	(*X*)
	Quota_Prelievo_Falda_X : LREAL;
	Quota_Deposito_Falda_SuCatastaPallet_X : LREAL;
	Quota_Deposito_Falda_SuPiazzola_X : LREAL;
	Quota_Fuori_Ingombro_X : LREAL;	
	
	(*Y*)
	Quota_Prelievo_Falda_Y 					: LREAL;
	Quota_Deposito_Falda_SuCatastaPallet_Y 	: LREAL;
	Quota_Deposito_Falda_SuPiazzola_Y		: LREAL;
	
	Quota_Fuori_Ingombro_Y					: LREAL;
	
	(*Z*)
	Quota_StartLenta_Prelievo_Falda_Z 					: LREAL;
	Quota_Prelievo_Falda_Z 								: LREAL;
	Quota_StartLenta_Deposito_Falda_SuPiazzola_Z 		: LREAL; //Se non si utilizza il tasteggio in fase di deposito si utilizza questa quota come quota di rilascio!!!
	Quota_Deposito_Falda_SuPiazzola_Z					: LREAL;
	Quota_StartLenta_Deposito_Falda_SuCatastaPallet_Z	: LREAL;
	Quota_Deposito_Falda_SuCatastaPallet_Z				: LREAL;
	QUota_Fuori_Ingombro_Falda_Z 						: LREAL;
	Quota_Attesa_Caduta_Falda_Z							: LREAL;
	
	(*k*)
	//Quota_Apertura_Prelievo_Falda_K : LREAL;
	//Quota_Chiusura_Prelievo_Falda_K : LREAL;
	//Quota_Apertura_Deposito_Falda_K : LREAL;
		
	(*J*)
	Quota_Rotazione_Prelievo_Falda 			: LREAL;
	Quota_Rotazione_Deposito_Falda 			: LREAL;
	
END_VAR
VAR_OUTPUT
	Inizializzato : BOOL;
END_VAR
VAR
	;	
END_VAR

(*
PRELIEVO FALDA:
1- Programma asse X per raggiungere magazzino falde da quota attuale in direzione X
2- Programma asse Y per raggiungere magazzino falde da quota attuale in direzione Y
3- Programma asse J per raggiungere l'angolo di rotazione richiesto
4- Programma asse K per raggiungere la quota di apertura pinza 
5- Programma asse Z per raggiungere la quota di cambio velocità in direzione Z (si passerà da veloce a lenta + tastatori disabilitati) in VELOCE
6- Programma asse Z in cui si effettua la traslazione in LENTA in direzione Z fino tocco dei tastatori
7- Programma asse K per raggiungere la quota di chiusura pinza !!!! PREVISTO MA NON UTILIZZATO !!!!!!

DEPOSITO FALDA:
8- Programma asse Z per raggiungere la quota di "Attesa caduta Falda" 
9- Programma asse Z per raggiungere la quota di "Fuori Ingombro" ostacoli 
10- Programma asse X per raggiungere la quota di deposito falda da quota attuale in direzione X; puù essere sul pallet in catasta(ciclo vuoti) o pallet su piazzola
11- Programma asse Y per posizione la quota di deposito falda da quota attuale in direzione Y
12: 
12.1- Programma asse Z per raggiungere la quota di rilascio falda in direzione Z su PIAZZOLA
12.2- Programma asse Z Z in cui si effettua la traslazione in LENTA in direzione Z fino tocco dei tastatori su CATASTA VUOTI

*)
Inizializzato := FALSE;
(*************************************************************************************************************************************)
(******************************************************  ASSE X **********************************************************************)
(*************************************************************************************************************************************)
(* Programma 51 Asse X : Traslazione Verso Postazione di Prelievo Pacco*)
Programma_X[X_PosPrelievoFalda].ID 					:= X_PosPrelievoFalda;
Programma_X[X_PosPrelievoFalda].Quota_Destinazione	:= Quota_Prelievo_Falda_X;
Programma_X[X_PosPrelievoFalda].Velocita			:= X_Par.Vel_Vuoto;
Programma_X[X_PosPrelievoFalda].Accelerazione		:= X_Par.Acc_Vuoto;
Programma_X[X_PosPrelievoFalda].Decelerazione		:= X_Par.Dec_Vuoto;
Programma_X[X_PosPrelievoFalda].Jerk				:= X_Par.Jerk_Vuoto;

(* Programma 52 Asse X : Traslazione Verso Postazione di deposito Falda su catasta vuoti*)
Programma_X[X_PosDepositoSuCatastaFalda].ID 					:= X_PosDepositoSuCatastaFalda;
Programma_X[X_PosDepositoSuCatastaFalda].Quota_Destinazione	:= Quota_Deposito_Falda_SuCatastaPallet_X;
Programma_X[X_PosDepositoSuCatastaFalda].Velocita			:= X_Par.Vel_Vuoto;
Programma_X[X_PosDepositoSuCatastaFalda].Accelerazione		:= X_Par.Acc_Vuoto;
Programma_X[X_PosDepositoSuCatastaFalda].Decelerazione		:= X_Par.Dec_Vuoto;
Programma_X[X_PosDepositoSuCatastaFalda].Jerk				:= X_Par.Jerk_Vuoto;

(* Programma 53 Asse X : Traslazione a quota di deposito Falda su piazzola*)
Programma_X[X_PosDepositoFalda].ID 					:= X_PosDepositoFalda;
Programma_X[X_PosDepositoFalda].Quota_Destinazione	:= Quota_Deposito_Falda_SuPiazzola_X;
Programma_X[X_PosDepositoFalda].Velocita			:= X_Par.Vel_Vuoto;
Programma_X[X_PosDepositoFalda].Accelerazione		:= X_Par.Acc_Vuoto;
Programma_X[X_PosDepositoFalda].Decelerazione		:= X_Par.Dec_Vuoto;
Programma_X[X_PosDepositoFalda].Jerk				:= X_Par.Jerk_Vuoto;

(* Programma 56 Asse Y : Traslazione a quota di riposo a Vuoto *)
Programma_X[X_PosFuoriIngombroVuotoFalda].ID 					:= X_PosFuoriIngombroVuotoFalda;
Programma_X[X_PosFuoriIngombroVuotoFalda].Quota_Destinazione	:= Quota_Fuori_Ingombro_X;
Programma_X[X_PosFuoriIngombroVuotoFalda].Velocita			:= X_Par.Vel_Vuoto;
Programma_X[X_PosFuoriIngombroVuotoFalda].Accelerazione		:= X_Par.Acc_Vuoto;
Programma_X[X_PosFuoriIngombroVuotoFalda].Decelerazione		:= X_Par.Dec_Vuoto;
Programma_X[X_PosFuoriIngombroVuotoFalda].Jerk				:= X_Par.Jerk_Vuoto;

(*************************************************************************************************************************************)
(******************************************************  ASSE Y **********************************************************************)
(*************************************************************************************************************************************)
(* Programma 51 Asse Y : Traslazione a quota di Prelievo Falda*)
Programma_Y[Y_PosPrelievoFalda].ID 					:= Y_PosPrelievoFalda;
Programma_Y[Y_PosPrelievoFalda].Quota_Destinazione	:= Quota_Prelievo_Falda_Y;
Programma_Y[Y_PosPrelievoFalda].Velocita			:= Y_Par.Vel_Vuoto;
Programma_Y[Y_PosPrelievoFalda].Accelerazione		:= Y_Par.Acc_Vuoto;
Programma_Y[Y_PosPrelievoFalda].Decelerazione		:= Y_Par.Dec_Vuoto;
Programma_Y[Y_PosPrelievoFalda].Jerk				:= Y_Par.Jerk_Vuoto;

(* Programma 52 Asse Y : Traslazione a quota di Deposito Falda su catasta vuoti*)
Programma_Y[Y_PosDepositoSuCatastaFalda].ID 					:= Y_PosDepositoSuCatastaFalda;
Programma_Y[Y_PosDepositoSuCatastaFalda].Quota_Destinazione	:= Quota_Deposito_Falda_SuCatastaPallet_Y;
Programma_Y[Y_PosDepositoSuCatastaFalda].Velocita			:= Y_Par.Vel_Vuoto;
Programma_Y[Y_PosDepositoSuCatastaFalda].Accelerazione		:= Y_Par.Acc_Vuoto;
Programma_Y[Y_PosDepositoSuCatastaFalda].Decelerazione		:= Y_Par.Dec_Vuoto;
Programma_Y[Y_PosDepositoSuCatastaFalda].Jerk				:= Y_Par.Jerk_Vuoto;

(* Programma 53 Asse Y : Traslazione a quota di Deposito Falda su piazzola*)
Programma_Y[Y_PosDepositoFalda].ID 					:= Y_PosDepositoFalda;
Programma_Y[Y_PosDepositoFalda].Quota_Destinazione	:= Quota_Deposito_Falda_SuPiazzola_Y;
Programma_Y[Y_PosDepositoFalda].Velocita			:= Y_Par.Vel_Vuoto;
Programma_Y[Y_PosDepositoFalda].Accelerazione		:= Y_Par.Acc_Vuoto;
Programma_Y[Y_PosDepositoFalda].Decelerazione		:= Y_Par.Dec_Vuoto;
Programma_Y[Y_PosDepositoFalda].Jerk				:= Y_Par.Jerk_Vuoto;

(* Programma 56 Asse Y : Traslazione a quota di riposo a Vuoto *)
Programma_Y[Y_PosFuoriIngombroVuotoFalda].ID 					:= Y_PosFuoriIngombroVuotoFalda;
Programma_Y[Y_PosFuoriIngombroVuotoFalda].Quota_Destinazione	:= Quota_Fuori_Ingombro_Y;
Programma_Y[Y_PosFuoriIngombroVuotoFalda].Velocita			:= Y_Par.Vel_Vuoto;
Programma_Y[Y_PosFuoriIngombroVuotoFalda].Accelerazione		:= Y_Par.Acc_Vuoto;
Programma_Y[Y_PosFuoriIngombroVuotoFalda].Decelerazione		:= Y_Par.Dec_Vuoto;
Programma_Y[Y_PosFuoriIngombroVuotoFalda].Jerk				:= Y_Par.Jerk_Vuoto;

(* Programma 66 Asse Y : Traslazione a quota di riposo con carico*)
Programma_Y[Y_PosFuoriIngombroCaricoFalda].ID 					:= Y_PosFuoriIngombroCaricoFalda;
Programma_Y[Y_PosFuoriIngombroCaricoFalda].Quota_Destinazione	:= Quota_Fuori_Ingombro_Y;
Programma_Y[Y_PosFuoriIngombroCaricoFalda].Velocita			:= Y_Par.Vel_Carico;
Programma_Y[Y_PosFuoriIngombroCaricoFalda].Accelerazione		:= Y_Par.Acc_Carico;
Programma_Y[Y_PosFuoriIngombroCaricoFalda].Decelerazione		:= Y_Par.Dec_Carico;
Programma_Y[Y_PosFuoriIngombroCaricoFalda].Jerk				:= Y_Par.Jerk_Carico;

(*************************************************************************************************************************************)
(******************************************************  ASSE Z **********************************************************************)
(*************************************************************************************************************************************)

(* Programma 51 Asse Z : Traslazione veloce fino alla quota ammessa in fase di Prelievo Falda*)
Programma_Z[Z_PosStartLentaPrelievoFalda].ID 					:= Z_PosStartLentaPrelievoFalda;
Programma_Z[Z_PosStartLentaPrelievoFalda].Quota_Destinazione	:= Quota_StartLenta_Prelievo_Falda_Z;
Programma_Z[Z_PosStartLentaPrelievoFalda].Velocita			:= Z_Par.Vel_Vuoto;
Programma_Z[Z_PosStartLentaPrelievoFalda].Accelerazione		:= Z_Par.Acc_Vuoto;
Programma_Z[Z_PosStartLentaPrelievoFalda].Decelerazione		:= Z_Par.Dec_Vuoto;
Programma_Z[Z_PosStartLentaPrelievoFalda].Jerk				:= Z_Par.Jerk_Vuoto;
Programma_Z[Z_PosStartLentaPrelievoFalda].DisabilitaTasteggio	:= TRUE;

(* Programma 52 Asse Z : Traslazione lenta fino al raggiungimento dei tastatori pinza*)
Programma_Z[Z_PosPrelievoInLentaFalda].ID 					:= Z_PosPrelievoInLentaFalda;
Programma_Z[Z_PosPrelievoInLentaFalda].Quota_Destinazione	:= Quota_Prelievo_Falda_Z;
Programma_Z[Z_PosPrelievoInLentaFalda].Velocita				:= Z_Par.Vel_Ridotta;
Programma_Z[Z_PosPrelievoInLentaFalda].Accelerazione		:= Z_Par.Acc_Vuoto;
Programma_Z[Z_PosPrelievoInLentaFalda].Decelerazione		:= Z_Par.Dec_Vuoto;
Programma_Z[Z_PosPrelievoInLentaFalda].Jerk					:= Z_Par.Jerk_Vuoto;
Programma_Z[Z_PosPrelievoInLentaFalda].DisabilitaTasteggio	:= FALSE;
Programma_Z[Z_PosPrelievoInLentaFalda].InnestoDiretto		:= TRUE;

(* Programma 53 Asse Z : Traslazione a quota di "Attesa caduta Falda"*)
Programma_Z[Z_PosAttesaCadutaFalda].ID 					:= Z_PosAttesaCadutaFalda;
Programma_Z[Z_PosAttesaCadutaFalda].Quota_Destinazione	:= Quota_Attesa_Caduta_Falda_Z;
Programma_Z[Z_PosAttesaCadutaFalda].Velocita			:= Z_Par.Vel_Ridotta;
Programma_Z[Z_PosAttesaCadutaFalda].Accelerazione		:= Z_Par.Acc_Vuoto;
Programma_Z[Z_PosAttesaCadutaFalda].Decelerazione		:= Z_Par.Dec_Vuoto;
Programma_Z[Z_PosAttesaCadutaFalda].Jerk				:= Z_Par.Jerk_Vuoto;
Programma_Z[Z_PosAttesaCadutaFalda].DisabilitaTasteggio	:= FALSE;

(* Programma 54 Asse Z : Traslazione a quota di "Fuori Ingombro"*)
Programma_Z[Z_PosFuoriIngombroFalda].ID 					:= Z_PosFuoriIngombroFalda;
Programma_Z[Z_PosFuoriIngombroFalda].Quota_Destinazione	:= Quota_Fuori_Ingombro_Falda_Z;
Programma_Z[Z_PosFuoriIngombroFalda].Velocita			:= Z_Par.Vel_Vuoto;
Programma_Z[Z_PosFuoriIngombroFalda].Accelerazione		:= Z_Par.Acc_Vuoto;
Programma_Z[Z_PosFuoriIngombroFalda].Decelerazione		:= Z_Par.Dec_Vuoto;
Programma_Z[Z_PosFuoriIngombroFalda].Jerk				:= Z_Par.Jerk_Vuoto;
Programma_Z[Z_PosFuoriIngombroFalda].DisabilitaTasteggio	:= TRUE;
Programma_Z[Z_PosFuoriIngombroFalda].InnestoDiretto		:= TRUE;

(* Programma 55 Asse Z : Traslazione veloce fino alla quota per deposito su catasta vuoti Pallet*)
Programma_Z[Z_PosStartLentaDepositoSuCatasta].ID 					:= Z_PosStartLentaDepositoSuCatasta;
Programma_Z[Z_PosStartLentaDepositoSuCatasta].Quota_Destinazione	:= Quota_StartLenta_Deposito_Falda_SuCatastaPallet_Z;
Programma_Z[Z_PosStartLentaDepositoSuCatasta].Velocita			:= Z_Par.Vel_Vuoto;
Programma_Z[Z_PosStartLentaDepositoSuCatasta].Accelerazione		:= Z_Par.Acc_Vuoto;
Programma_Z[Z_PosStartLentaDepositoSuCatasta].Decelerazione		:= Z_Par.Dec_Vuoto;
Programma_Z[Z_PosStartLentaDepositoSuCatasta].Jerk				:= Z_Par.Jerk_Vuoto;
Programma_Z[Z_PosStartLentaDepositoSuCatasta].DisabilitaTasteggio	:= TRUE;
	
(* Programma 56 Asse Z : Traslazione lenta fino al raggiungimento dei tastatori pinza deposito su catasta vuoti Pallet*)
Programma_Z[Z_PosDepositoInLentaSuCatasta].ID 					:= Z_PosDepositoInLentaSuCatasta;
Programma_Z[Z_PosDepositoInLentaSuCatasta].Quota_Destinazione	:= Quota_Deposito_Falda_SuCatastaPallet_Z;
Programma_Z[Z_PosDepositoInLentaSuCatasta].Velocita			:= Z_Par.Vel_Ridotta;
Programma_Z[Z_PosDepositoInLentaSuCatasta].Accelerazione		:= Z_Par.Acc_Vuoto;
Programma_Z[Z_PosDepositoInLentaSuCatasta].Decelerazione		:= Z_Par.Dec_Vuoto;
Programma_Z[Z_PosDepositoInLentaSuCatasta].Jerk				:= Z_Par.Jerk_Vuoto;
Programma_Z[Z_PosDepositoInLentaSuCatasta].DisabilitaTasteggio	:= FALSE;
Programma_Z[Z_PosDepositoInLentaSuCatasta].InnestoDiretto		:= TRUE;

(* Programma 57 Asse Z : Traslazione veloce fino alla quota per deposito su postazione*)
Programma_Z[Z_PosStartLentaDepositoFalda].ID 					:= Z_PosStartLentaDepositoFalda;
Programma_Z[Z_PosStartLentaDepositoFalda].Quota_Destinazione	:= Quota_StartLenta_Deposito_Falda_SuPiazzola_Z;
Programma_Z[Z_PosStartLentaDepositoFalda].Velocita			:= Z_Par.Vel_Vuoto;
Programma_Z[Z_PosStartLentaDepositoFalda].Accelerazione		:= Z_Par.Acc_Vuoto;
Programma_Z[Z_PosStartLentaDepositoFalda].Decelerazione		:= Z_Par.Dec_Vuoto;
Programma_Z[Z_PosStartLentaDepositoFalda].Jerk				:= Z_Par.Jerk_Vuoto;
Programma_Z[Z_PosStartLentaDepositoFalda].DisabilitaTasteggio	:= TRUE;
	
(* Programma 58 Asse Z : Traslazione lenta fino al raggiungimento dei tastatori pinza *)
Programma_Z[Z_PosDepositoInLentaFalda].ID 					:= Z_PosDepositoInLentaFalda;
Programma_Z[Z_PosDepositoInLentaFalda].Quota_Destinazione	:= Quota_Deposito_Falda_SuPiazzola_Z;
Programma_Z[Z_PosDepositoInLentaFalda].Velocita				:= Z_Par.Vel_Ridotta;
Programma_Z[Z_PosDepositoInLentaFalda].Accelerazione		:= Z_Par.Acc_Vuoto;
Programma_Z[Z_PosDepositoInLentaFalda].Decelerazione		:= Z_Par.Dec_Vuoto;
Programma_Z[Z_PosDepositoInLentaFalda].Jerk					:= Z_Par.Jerk_Vuoto;
Programma_Z[Z_PosDepositoInLentaFalda].DisabilitaTasteggio	:= FALSE;

(*
(*************************************************************************************************************************************)
(******************************************************  ASSE K **********************************************************************)
(*************************************************************************************************************************************)
(* Programma 51 Asse K : Apertura pinza per prelievo falda *)
Programma_K[51].ID 					:= 51;
Programma_K[51].Quota_Destinazione	:= Quota_Apertura_Prelievo_Falda_K;
Programma_K[51].Velocita			:= K_Par.Vel_Vuoto;
Programma_K[51].Accelerazione		:= K_Par.Acc_Vuoto;
Programma_K[51].Decelerazione		:= K_Par.Dec_Vuoto;
Programma_K[51].Jerk				:= K_Par.Jerk_Vuoto;
Programma_K[51].Torque				:= 100;
(* Programma 52 Asse K : Chiusura pinza per falda prelievo *)
Programma_K[52].ID 					:= 52;
Programma_K[52].Quota_Destinazione	:= Quota_Chiusura_Prelievo_Falda_K;
Programma_K[52].Velocita			:= K_Par.Vel_Vuoto;
Programma_K[52].Accelerazione		:= K_Par.Acc_Vuoto;
Programma_K[52].Decelerazione		:= K_Par.Dec_Vuoto;
Programma_K[52].Jerk				:= K_Par.Jerk_Vuoto;
Programma_K[52].Torque				:= 100;

(* Programma 53 Asse K : Apertura pinza per deposito falda *)
Programma_K[53].ID 					:= 53;
Programma_K[53].Quota_Destinazione	:= Quota_Apertura_Deposito_Falda_K;
Programma_K[53].Velocita			:= K_Par.Vel_Vuoto;
Programma_K[53].Accelerazione		:= K_Par.Acc_Vuoto;
Programma_K[53].Decelerazione		:= K_Par.Dec_Vuoto;
Programma_K[53].Jerk				:= K_Par.Jerk_Vuoto;
Programma_K[53].Torque				:= 100;
*)

(*************************************************************************************************************************************)
(******************************************************  ASSE J **********************************************************************)
(*************************************************************************************************************************************)

(* Programma 10 Asse J : Rotazione a quota pelievo falda *)
Programma_J[10].ID 					:= 10;
Programma_J[10].Quota_Destinazione	:= Quota_Rotazione_Prelievo_Falda;
Programma_J[10].Velocita			:= J_Par.Vel_Vuoto;
Programma_J[10].Accelerazione		:= J_Par.Acc_Vuoto;
Programma_J[10].Decelerazione		:= J_Par.Dec_Vuoto;
Programma_J[10].Jerk				:= J_Par.Jerk_Vuoto;

(* Programma 11 Asse J : Rotazione a quota deposito falda *)
Programma_J[11].ID 					:= 11;
Programma_J[11].Quota_Destinazione	:= Quota_Rotazione_Deposito_Falda;
Programma_J[11].Velocita			:= J_Par.Vel_Carico;
Programma_J[11].Accelerazione		:= J_Par.Acc_Carico;
Programma_J[11].Decelerazione		:= J_Par.Dec_Carico;
Programma_J[11].Jerk				:= J_Par.Jerk_Carico;

Inizializzato := TRUE;

END_FUNCTION_BLOCK

// ---- POUs/TFCicliDiLavoro/ProgrammiMovimento/TFProgramma_Ciclo_Lastra.TcPOU
FUNCTION_BLOCK TFProgramma_Ciclo_Lastra
VAR_INPUT
	X_Par : Ax_Program_Parameters; // Parametri degli assi
	Y_Par : Ax_Program_Parameters; // Parametri degli assi
	Z_Par : Ax_Program_Parameters; // Parametri degli assi
	//K_Par : Ax_Program_Parameters; // Parametri degli assi
	J_Par : Ax_Program_Parameters; // Parametri degli assi
	
	(*X*)
	Quota_Prelievo_Lastra_X 			: LREAL;
	Quota_StartLenta_Prelievo_Lastra_X 	: LREAL;	// quota approccio
	Quota_Deposito_Lastra_X 			: LREAL;
	Quota_StartLenta_Deposito_Lastra_X 	: LREAL;	// quota approccio
	Quota_Distacco_Lastra_X 			: LREAL; 	//Quota di distacco lastra
	Quota_Fuori_Ingombro_SenzaCarico_X 	: LREAL; 
	Quota_Fuori_Ingombro_Carico_X 		: LREAL;
	Quota_PosGiroPiezaTraCavalleteX     : LREAL;   //Cuota Posicion Giro Trabajo Cavallete
	(*Y*)
	Quota_Prelievo_Lastra_Y 				: LREAL; // Quota di prelievo lastra
	Quota_StartLenta_Prelievo_Lastra_Y 		: LREAL; // quota approccio in prelievo
	Quota_StartLenta_Deposito_Lastra_Y 		: LREAL; // quota approccio in deposito
	Quota_Deposito_Lastra_Y 				: LREAL; // Quota deposito lastra 
	Quota_Fuori_Ingombro_Y 					: LREAL; // Quota Fuori ingombro in fase di prelievo
	Quota_Distacco_Lastra_Y 				: LREAL; // Quota a cui si posiziona in fase di distacco lastra
	Quota_Posicion_Giro_Pinza				: LREAL; // Quota posicion giro pieza para cavalina EjeX
	Quota_PasilloCavallete0GradosY          : LREAL ;
	Quota_PasilloCavallete1800GradosY       : LREAL ;

	(*Z*)
	Quota_StartLenta_Prelievo_Lastra_Z 		: LREAL;
	Quota_Prelievo_Lastra_Z 				: LREAL;
	Quota_StartLenta_Deposito_Lastra_Z 		: LREAL; // quota approccio
	Quota_Deposito_Lastra_Z 				: LREAL;
	Quota_Fuori_Ingombro_ConCarico_Z		: LREAL;
	Quota_Fuori_Ingombro_SenzaCarico_Z 		: LREAL;
	DisabilitaDepositoConTasteggio 			: BOOL;
	Quota_Distacco_Lastra_Z		 			: LREAL; //Quota di distacco lastra
	Quota_PostScarico							: LREAL;//posizione che si porta dopo aver scaricato la lastra
	
	(*J*)
	Quota_Rotazione_Prelievo_Lastra 			: LREAL;
	Quota_Rotazione_Deposito_Lastra 			: LREAL;
	Quota_Rotazione_StartTasteggio_Lastra 		: LREAL;
	Quota_Fuori_Ingombro_J						: LREAL;
	Quota_Rotazione_Sfogliatura					: LREAL;
	Quota_PostScaricoJ						: LREAL;//posizione che si porta dopo aver scaricato la lastra
	Quota_Fuori_Ingombro_AttualeJ			: LREAL;

	
END_VAR
VAR_OUTPUT
	Inizializzato : BOOL;
END_VAR
VAR
	;	
END_VAR

(*
X:
(* Programma 1 Asse X : Traslazione Verso Postazione di Prelievo Lastra*)
(* Programma 2 Asse X : Traslazione veloce a quota ammessa per veloce di deposito Pacco su piazzola*)
(* Programma 3 Asse X : Traslazione lenta a quota di deposito Pacco su piazzola*)
Y:
(* Programma 1 Asse Y : Traslazione a quota di Prelievo Pacco*)
(* Programma 2 Asse Y : Traslazione veloce a quota ammessa per veloce per Deposito Pacco su piazzola*)
(* Programma 3 Asse Y : Traslazione a quota di Deposito Pacco su piazzola*)

Z:
(* Programma 1 Asse Z : Traslazione veloce fino alla quota ammessa in veloce in fase di Prelievo pacco*)
(* Programma 2 Asse Z : Traslazione lenta fino al raggiungimento della quota di prelievo*)
(* Programma 3 Asse Z : Traslazione veloce fino alla quota ammessa in veloce in fase di deposito pacco *)
(* Programma 4 Asse Z : Traslazione lenta fino alla quota di deposito su piazzola*)
(* Programma 5 Asse Z : Traslazione a quota di "Fuori Ingombro" con carico a bordo*)
(* Programma 6 Asse Z : Traslazione a quota di "Fuori Ingombro" con carico a bordo*)

J:
(* Programma 0 Asse J : Rotazione 90° a vuoto *)
(* Programma 1 Asse J : Rotazione 0° a vuoto *)
(* Programma 2 Asse J : Rotazione 180° a vuoto *)
(* Programma 3 Asse J : Rotazione 270° a vuoto *)
(* Programma 4 Asse J : Rotazione 90° con carico *)
(* Programma 5 Asse J : Rotazione 0° con carico *)
(* Programma 6 Asse J : Rotazione 180° con carico *)
(* Programma 7 Asse J : Rotazione 270° con carico *)
*)
Inizializzato := FALSE;
(*************************************************************************************************************************************)
(******************************************************  ASSE X **********************************************************************)
(*************************************************************************************************************************************)
(* Programma 101 Asse X : Traslazione veloce Verso Postazione di Prelievo in quoata di start lenta *)
Programma_X[101].ID 				:= 101;
Programma_X[101].Quota_Destinazione	:= Quota_StartLenta_Prelievo_Lastra_X;
Programma_X[101].Velocita			:= X_Par.Vel_Vuoto;
Programma_X[101].Accelerazione		:= X_Par.Acc_Vuoto;
Programma_X[101].Decelerazione		:= X_Par.Dec_Vuoto;
Programma_X[101].Jerk				:= X_Par.Jerk_Vuoto;

(* Programma 102 Asse X : Traslazione in lenta fino alla posizione di prelievo*)
Programma_X[102].ID 				:= 102;
Programma_X[102].Quota_Destinazione	:= Quota_Prelievo_Lastra_X;
Programma_X[102].Velocita			:= X_Par.Vel_Ridotta;
Programma_X[102].Accelerazione		:= X_Par.Acc_Vuoto;
Programma_X[102].Decelerazione		:= X_Par.Dec_Vuoto;
Programma_X[102].Jerk				:= X_Par.Jerk_Vuoto;

(* Programma 103 Asse X : Traslazione in lenta per distacco della lastra *)
Programma_X[103].ID 				:= 103;
Programma_X[103].Quota_Destinazione	:= Quota_Distacco_Lastra_X;
Programma_X[103].Velocita			:= X_Par.Vel_Ridotta;
Programma_X[103].Accelerazione		:= X_Par.Acc_Carico;
Programma_X[103].Decelerazione		:= X_Par.Dec_Carico;
Programma_X[103].Jerk				:= X_Par.Jerk_Carico;
Programma_X[103].InnestoDiretto		:= TRUE;

(* Programma 104 Asse X : Traslazione veloce alla quota di approccio in deposito *)
Programma_X[104].ID 				:= 104;
Programma_X[104].Quota_Destinazione	:= Quota_StartLenta_Deposito_Lastra_X;
Programma_X[104].Velocita			:= X_Par.Vel_Carico;
Programma_X[104].Accelerazione		:= X_Par.Acc_Carico;
Programma_X[104].Decelerazione		:= X_Par.Dec_Carico;
Programma_X[104].Jerk				:= X_Par.Jerk_Carico;
Programma_X[104].InnestoDiretto		:= TRUE;

(* Programma 105 Asse X : Traslazione LENTA alla quota di deposito *)
Programma_X[105].ID 				:= 105;
Programma_X[105].Quota_Destinazione	:= Quota_Deposito_Lastra_X;
Programma_X[105].Velocita			:= X_Par.Vel_Ridotta;
Programma_X[105].Accelerazione		:= X_Par.Acc_Carico;
Programma_X[105].Decelerazione		:= X_Par.Dec_Carico;
Programma_X[105].Jerk				:= X_Par.Jerk_Carico;
Programma_X[105].InnestoDiretto		:= TRUE;

(* Programma 106 Asse X : Traslazione a quota di "Fuori Ingombro" senza carico a bordo*)
Programma_X[106].ID 				:= 106;
Programma_X[106].Quota_Destinazione	:= Quota_Fuori_Ingombro_SenzaCarico_X;
Programma_X[106].Velocita			:= X_Par.Vel_Vuoto;
Programma_X[106].Accelerazione		:= X_Par.Acc_Vuoto;
Programma_X[106].Decelerazione		:= X_Par.Dec_Vuoto;
Programma_X[106].Jerk					:= X_Par.Jerk_Vuoto;
Programma_X[106].DisabilitaTasteggio	:= TRUE;

(* Programma 126 Asse X : Traslazione a quota di "Fuori Ingombro" poso con carico*)
Programma_X[126].ID 				:= 126;
Programma_X[126].Quota_Destinazione	:= Quota_Fuori_Ingombro_Carico_X;
Programma_X[126].Velocita			:= X_Par.Vel_Carico;
Programma_X[126].Accelerazione		:= X_Par.Acc_Carico;
Programma_X[126].Decelerazione		:= X_Par.Dec_Carico;
Programma_X[126].Jerk				:= X_Par.Jerk_Carico;

(* Programma 127 Asse X : Traslazione a quota posicion Para invertir guiro*)
Programma_X[X_PosGiroPiezaTraCavallete].ID 				:= 127;
Programma_X[X_PosGiroPiezaTraCavallete].Quota_Destinazione	:= Quota_PosGiroPiezaTraCavalleteX;
Programma_X[X_PosGiroPiezaTraCavallete].Velocita			:= X_Par.Vel_Carico;
Programma_X[X_PosGiroPiezaTraCavallete].Accelerazione		:= X_Par.Acc_Carico;
Programma_X[X_PosGiroPiezaTraCavallete].Decelerazione		:= X_Par.Dec_Carico;
Programma_X[X_PosGiroPiezaTraCavallete].Jerk				:= X_Par.Jerk_Carico;

(*************************************************************************************************************************************)
(******************************************************  ASSE Y **********************************************************************)
(*************************************************************************************************************************************)
(* Programma 101 Asse Y : Traslazione veloce Verso Postazione di Prelievo in quoata di start lenta *)
Programma_Y[101].ID 				:= 101;
Programma_Y[101].Quota_Destinazione	:= Quota_StartLenta_Prelievo_Lastra_Y;
Programma_Y[101].Velocita			:= Y_Par.Vel_Vuoto;
Programma_Y[101].Accelerazione		:= Y_Par.Acc_Vuoto;
Programma_Y[101].Decelerazione		:= Y_Par.Dec_Vuoto;
Programma_Y[101].Jerk				:= Y_Par.Jerk_Vuoto;
Programma_Y[101].DisabilitaTasteggio	:= FALSE;

(* Programma 102 Asse Y : Traslazione in lenta fino alla posizione di prelievo*)
Programma_Y[102].ID 				:= 102;
Programma_Y[102].Quota_Destinazione	:= Quota_Prelievo_Lastra_Y;
Programma_Y[102].Velocita			:= Y_Par.Vel_Ridotta;
Programma_Y[102].Accelerazione		:= Y_Par.Acc_Carico;
Programma_Y[102].Decelerazione		:= Y_Par.Dec_Carico;
Programma_Y[102].Jerk				:= Y_Par.Jerk_Carico;
//Programma_Y[102].DisabilitaTasteggio	:= FALSE;
Programma_Y[102].DisabilitaTasteggio	:= TRUE;

(* Programma 103 Asse Y : Traslazione in lenta per distacco della lastra *)
Programma_Y[103].ID 				:= 103;
Programma_Y[103].Quota_Destinazione	:= Quota_Distacco_Lastra_Y;
Programma_Y[103].Velocita			:= Y_Par.Vel_Ridotta;
Programma_Y[103].Accelerazione		:= Y_Par.Acc_Carico;
Programma_Y[103].Decelerazione		:= Y_Par.Dec_Carico;
Programma_Y[103].Jerk				:= Y_Par.Jerk_Carico;
Programma_Y[103].InnestoDiretto		:= TRUE;

(* Programma 104 Asse Y : Traslazione veloce alla quota di approccio in deposito *)
Programma_Y[104].ID 				:= 104;
Programma_Y[104].Quota_Destinazione	:= Quota_StartLenta_Deposito_Lastra_Y;
Programma_Y[104].Velocita			:= Y_Par.Vel_Carico;
Programma_Y[104].Accelerazione		:= Y_Par.Acc_Carico;
Programma_Y[104].Decelerazione		:= Y_Par.Dec_Carico;
Programma_Y[104].Jerk				:= Y_Par.Jerk_Carico;
Programma_Y[104].InnestoDiretto		:= TRUE;
Programma_Y[104].DisabilitaTasteggio := FALSE;

(* Programma 105 Asse Y : Traslazione LENTA alla quota di deposito *)
Programma_Y[105].ID 				:= 105;
Programma_Y[105].Quota_Destinazione	:= Quota_Deposito_Lastra_Y;
Programma_Y[105].Velocita			:= Y_Par.Vel_Ridotta;
Programma_Y[105].Accelerazione		:= Y_Par.Acc_Carico;
Programma_Y[105].Decelerazione		:= Y_Par.Dec_Carico;
Programma_Y[105].Jerk				:= Y_Par.Jerk_Carico;
Programma_Y[105].InnestoDiretto		:= TRUE;
Programma_Y[105].DisabilitaTasteggio	:= FALSE;

(* Programma 6 Asse Y : Traslazione a quota "Fuori Ingombro"  a Vuoto *)
Programma_Y[106].ID 				:= 106;
Programma_Y[106].Quota_Destinazione	:= Quota_Fuori_Ingombro_Y;
Programma_Y[106].Velocita			:= Y_Par.Vel_Vuoto;
Programma_Y[106].Accelerazione		:= Y_Par.Acc_Vuoto;
Programma_Y[106].Decelerazione		:= Y_Par.Dec_Vuoto;
Programma_Y[106].Jerk				:= Y_Par.Jerk_Vuoto;
Programma_Y[106].DisabilitaTasteggio	:= TRUE;
(* Programma 126 Asse Y : Traslazione a quota "Fuori Ingombro" con carico*)
Programma_Y[126].ID 				:= 126;
Programma_Y[126].Quota_Destinazione	:= Quota_Fuori_Ingombro_Y;
Programma_Y[126].Velocita			:= Y_Par.Vel_Carico;
Programma_Y[126].Accelerazione		:= Y_Par.Acc_Carico;
Programma_Y[126].Decelerazione		:= Y_Par.Dec_Carico;
Programma_Y[126].Jerk				:= Y_Par.Jerk_Carico;
Programma_Y[126].DisabilitaTasteggio	:= TRUE;

(* Programma 127 Asse Y : Traslazione a quota "Possicion Girar Pieza " con carico*)
Programma_Y[127].ID 				:= 127;
Programma_Y[127].Quota_Destinazione	:= Quota_Posicion_Giro_Pinza;
Programma_Y[127].Velocita			:= Y_Par.Vel_Carico;
Programma_Y[127].Accelerazione		:= Y_Par.Acc_Carico;
Programma_Y[127].Decelerazione		:= Y_Par.Dec_Carico;
Programma_Y[127].Jerk				:= Y_Par.Jerk_Carico;
Programma_Y[127].DisabilitaTasteggio	:= TRUE;

(* Programma 128 Asse Y : Traslazione a quota "Possicion Girar Pieza " con carico*)
Programma_Y[Y_PosPasillo0grados].ID 					:= Y_PosPasillo0grados;
Programma_Y[Y_PosPasillo0grados].Quota_Destinazione		:= Quota_PasilloCavallete0GradosY;
Programma_Y[Y_PosPasillo0grados].Velocita				:= Y_Par.Vel_Carico;
Programma_Y[Y_PosPasillo0grados].Accelerazione			:= Y_Par.Acc_Carico;
Programma_Y[Y_PosPasillo0grados].Decelerazione			:= Y_Par.Dec_Carico;
Programma_Y[Y_PosPasillo0grados].Jerk					:= Y_Par.Jerk_Carico;
Programma_Y[Y_PosPasillo0grados].DisabilitaTasteggio	:= TRUE;

(* Programma 129 Asse Y : Traslazione a quota "Possicion Girar Pieza " con carico*)
Programma_Y[Y_PosPasillo180grados].ID 					:= Y_PosPasillo180grados;
Programma_Y[Y_PosPasillo180grados].Quota_Destinazione	:= Quota_PasilloCavallete1800GradosY;
Programma_Y[Y_PosPasillo180grados].Velocita				:= Y_Par.Vel_Carico;
Programma_Y[Y_PosPasillo180grados].Accelerazione		:= Y_Par.Acc_Carico;
Programma_Y[Y_PosPasillo180grados].Decelerazione		:= Y_Par.Dec_Carico;
Programma_Y[Y_PosPasillo180grados].Jerk					:= Y_Par.Jerk_Carico;
Programma_Y[Y_PosPasillo180grados].DisabilitaTasteggio	:= TRUE;

(*************************************************************************************************************************************)
(******************************************************  ASSE Z **********************************************************************)
(*************************************************************************************************************************************)

(* Programma 101 Asse Z : Traslazione veloce Verso Postazione di Prelievo in quoata di start lenta *)
Programma_Z[101].ID 					:= 101;
Programma_Z[101].Quota_Destinazione		:= Quota_StartLenta_Prelievo_Lastra_Z;
Programma_Z[101].Velocita				:= Z_Par.Vel_Vuoto;
Programma_Z[101].Accelerazione			:= Z_Par.Acc_Vuoto;
Programma_Z[101].Decelerazione			:= Z_Par.Dec_Vuoto;
Programma_Z[101].Jerk					:= Z_Par.Jerk_Vuoto;
Programma_Z[101].DisabilitaTasteggio	:= TRUE;

(* Programma 102 Asse Z : Traslazione in lenta fino alla posizione di prelievo*)
Programma_Z[102].ID 				:= 102;
Programma_Z[102].Quota_Destinazione	:= Quota_Prelievo_Lastra_Z;
Programma_Z[102].Velocita			:= Z_Par.Vel_Ridotta;
Programma_Z[102].Accelerazione		:= Z_Par.Acc_Vuoto;
Programma_Z[102].Decelerazione		:= Z_Par.Dec_Vuoto;
Programma_Z[102].Jerk					:= Z_Par.Jerk_Vuoto;
Programma_Z[102].DisabilitaTasteggio	:= FALSE;

(* Programma 103 Asse Z : Traslazione in lenta per distacco della lastra *)
Programma_Z[103].ID 				:= 103;
Programma_Z[103].Quota_Destinazione	:= Quota_Distacco_Lastra_Z;
Programma_Z[103].Velocita			:= MAX(2,HMI_VelocitaDistaccoLastra_Z);//Z_Par.Vel_Ridotta;
Programma_Z[103].Accelerazione		:= Z_Par.Acc_Carico;
Programma_Z[103].Decelerazione		:= Z_Par.Dec_Carico;
Programma_Z[103].Jerk				:= Z_Par.Jerk_Carico;
Programma_Z[103].DisabilitaTasteggio	:= TRUE;

(* Programma 104 Asse Z : Traslazione veloce alla quota di approccio in deposito *)
Programma_Z[104].ID 				:= 104;
Programma_Z[104].Quota_Destinazione	:= Quota_StartLenta_Deposito_Lastra_Z;
Programma_Z[104].Velocita			:= Z_Par.Vel_Carico;
Programma_Z[104].Accelerazione		:= Z_Par.Acc_Carico;
Programma_Z[104].Decelerazione		:= Z_Par.Dec_Carico;
Programma_Z[104].Jerk					:= Z_Par.Jerk_Carico;
Programma_Z[104].DisabilitaTasteggio	:= FALSE;//DisabilitaDepositoConTasteggio;
Programma_Z[104].InnestoDiretto		:= TRUE;

(* Programma 105 Asse Z : Traslazione lenta alla quota di deposito *)
Programma_Z[105].ID 					:= Z_PosDepositoInLentaLastra;
Programma_Z[105].Quota_Destinazione		:= Quota_Deposito_Lastra_Z;
Programma_Z[105].Velocita				:= Z_Par.Vel_Ridotta;
Programma_Z[105].Accelerazione			:= Z_Par.Acc_Carico;
Programma_Z[105].Decelerazione			:= Z_Par.Dec_Carico;
Programma_Z[105].Jerk					:= Z_Par.Jerk_Carico;
Programma_Z[105].DisabilitaTasteggio 	:= FALSE;//NOT HMI_AbilitaDepositoPaccoOrrizzontaleConTasteggio;

(* Programma 106 Asse Z : Traslazione a quota di "Fuori Ingombro" senza carico a bordo*)
Programma_Z[106].ID 				:= 106;
Programma_Z[106].Quota_Destinazione	:= Quota_Fuori_Ingombro_SenzaCarico_Z;
Programma_Z[106].Velocita			:= Z_Par.Vel_Vuoto;
Programma_Z[106].Accelerazione		:= Z_Par.Acc_Vuoto;
Programma_Z[106].Decelerazione		:= Z_Par.Dec_Vuoto;
Programma_Z[106].Jerk					:= Z_Par.Jerk_Vuoto;
Programma_Z[106].DisabilitaTasteggio	:= TRUE;

(* Programma 126 Asse Z : Traslazione a quota "Fuori Ingombro" con carico*)
Programma_Z[126].ID 				:= 126;
Programma_Z[126].Quota_Destinazione	:= Quota_Fuori_Ingombro_ConCarico_Z;
Programma_Z[126].Velocita			:= Z_Par.Vel_Carico;
Programma_Z[126].Accelerazione		:= Z_Par.Acc_Carico;
Programma_Z[126].Decelerazione		:= Z_Par.Dec_Carico;
Programma_Z[126].Jerk				:= Z_Par.Jerk_Carico;
Programma_Z[126].DisabilitaTasteggio	:= TRUE;
(* Programma 107 Asse Z : Traslazione a quota deposito pacco in veloce usato senza approccio*)
Programma_Z[107].ID 				:= 107;
Programma_Z[107].Quota_Destinazione	:= Quota_Deposito_Lastra_Z;
Programma_Z[107].Velocita			:= Z_Par.Vel_Carico;
Programma_Z[107].Accelerazione		:= Z_Par.Acc_Carico;
Programma_Z[107].Decelerazione		:= Z_Par.Dec_Carico;
Programma_Z[107].Jerk					:= Z_Par.Jerk_Carico;
Programma_Z[107].DisabilitaTasteggio	:= TRUE;

(* Programma 107 Asse Z : Traslazione a quota deposito pacco in veloce usato senza approccio*)
Programma_Z[Z_PosPostScarico].ID 				:= INT_TO_UINT(Z_PosPostScarico);
Programma_Z[Z_PosPostScarico].Quota_Destinazione	:= Quota_PostScarico;
Programma_Z[Z_PosPostScarico].Velocita			:= Z_Par.Vel_Carico;//Z_Par.Vel_Vuoto;
Programma_Z[Z_PosPostScarico].Accelerazione		:= Z_Par.Acc_Carico;
Programma_Z[Z_PosPostScarico].Decelerazione		:= Z_Par.Dec_Carico;
Programma_Z[Z_PosPostScarico].Jerk					:= Z_Par.Jerk_Carico;
Programma_Z[Z_PosPostScarico].DisabilitaTasteggio	:= TRUE;


(*
(*************************************************************************************************************************************)
(******************************************************  ASSE K **********************************************************************)
(*************************************************************************************************************************************)

(* Programma 101 Asse K : Apertura pinza per prelievo pacco *)
Programma_K[101].ID 				:= 101;
Programma_K[101].Quota_Destinazione	:= Quota_Apertura_Prelievo_Pacco_K;
Programma_K[101].Velocita			:= K_Par.Vel_Vuoto;
Programma_K[101].Accelerazione		:= K_Par.Acc_Vuoto;
Programma_K[101].Decelerazione		:= K_Par.Dec_Vuoto;
Programma_K[101].Jerk				:= K_Par.Jerk_Vuoto;
Programma_K[101].Torque				:= K_Par.Torque;
Programma_K[101].Controllo_Tastatori	:= TRUE;
Programma_K[101].ControlloCoppiaAbilitato := FALSE;


(* Programma 102 Asse K : Chiusura pinza per prelievo pacco *)
Programma_K[102].ID 				:= 102;
Programma_K[102].Quota_Destinazione	:= Quota_Chiusura_Prelievo_Pacco_K;
Programma_K[102].Velocita			:= K_Par.Vel_Vuoto;
Programma_K[102].Accelerazione		:= K_Par.Acc_Vuoto;
Programma_K[102].Decelerazione		:= K_Par.Dec_Vuoto;
Programma_K[102].Jerk				:= K_Par.Jerk_Vuoto;
Programma_K[102].Torque				:= K_Par.Torque;
Programma_K[102].Controllo_Tastatori	:= FALSE;
Programma_K[102].ControlloCoppiaAbilitato := Abilitazione_Controllo_Coppia_K;

(* Programma 103 Asse K : Apertura pinza per deposito pacco *)
Programma_K[103].ID 				:= 103;
Programma_K[103].Quota_Destinazione	:= Quota_Apertura_Deposito_Pacco_K;
Programma_K[103].Velocita			:= K_Par.Vel_Vuoto;
Programma_K[103].Accelerazione		:= K_Par.Acc_Vuoto;
Programma_K[103].Decelerazione		:= K_Par.Dec_Vuoto;
Programma_K[103].Jerk				:= K_Par.Jerk_Vuoto;
Programma_K[103].Torque				:= K_Par.Torque;
Programma_K[103].Controllo_Tastatori	:= TRUE;
Programma_K[103].ControlloCoppiaAbilitato := FALSE;
*)

(*************************************************************************************************************************************)
(******************************************************  ASSE J **********************************************************************)
(*************************************************************************************************************************************)
(*************************************************************************************************************************************)
(******************************************************  ASSE J **********************************************************************)
(*************************************************************************************************************************************)
(* Programma 6 Asse J : Traslazione a quota di FUORI INGOMBRO*)
Programma_J[J_PosFuoriIngombro].ID 					:= TO_UINT(J_PosFuoriIngombro);
Programma_J[J_PosFuoriIngombro].Quota_Destinazione	:= Quota_Fuori_Ingombro_J;
Programma_J[J_PosFuoriIngombro].Velocita			:= J_Par.Vel_Vuoto;
Programma_J[J_PosFuoriIngombro].Accelerazione		:= J_Par.Acc_Vuoto;
Programma_J[J_PosFuoriIngombro].Decelerazione		:= J_Par.Dec_Vuoto;
Programma_J[J_PosFuoriIngombro].Jerk				:= J_Par.Jerk_Vuoto;
Programma_J[J_PosFuoriIngombro].DisabilitaTasteggio	:= TRUE;

(* Programma 12 Asse J : Rotazione a quota di PRELIEVO LASTRA *)
Programma_J[J_PosPrelievoLastra].ID 					:= TO_UINT(J_PosPrelievoLastra);
Programma_J[J_PosPrelievoLastra].Quota_Destinazione	:= Quota_Rotazione_Prelievo_Lastra;
Programma_J[J_PosPrelievoLastra].Velocita			:= J_Par.Vel_Vuoto;
Programma_J[J_PosPrelievoLastra].Accelerazione		:= J_Par.Acc_Vuoto;
Programma_J[J_PosPrelievoLastra].Decelerazione		:= J_Par.Dec_Vuoto;
Programma_J[J_PosPrelievoLastra].Jerk				:= J_Par.Jerk_Vuoto;
Programma_J[J_PosPrelievoLastra].DisabilitaTasteggio	:= TRUE;

(* Programma 13 Asse J : Rotazione a quota di deposito DEPOSITO LASTRA *)
Programma_J[J_PosDepositoLastra].ID 				:= TO_UINT(J_PosDepositoLastra);
Programma_J[J_PosDepositoLastra].Quota_Destinazione	:= Quota_Rotazione_Deposito_Lastra;
Programma_J[J_PosDepositoLastra].Velocita			:= J_Par.Vel_Carico;
Programma_J[J_PosDepositoLastra].Accelerazione		:= J_Par.Acc_Carico;
Programma_J[J_PosDepositoLastra].Decelerazione		:= J_Par.Dec_Carico;
Programma_J[J_PosDepositoLastra].Jerk				:= J_Par.Jerk_Carico;
Programma_J[J_PosDepositoLastra].DisabilitaTasteggio	:= TRUE;

(* Programma 14 Asse J : Rotazione a quota di START APPROCCIO per prelievo su cavallina *)
Programma_J[J_PosStartApproccioPrelLastra].ID 					:= TO_UINT(J_PosStartApproccioPrelLastra);
Programma_J[J_PosStartApproccioPrelLastra].Quota_Destinazione	:= Quota_Rotazione_StartTasteggio_Lastra;
Programma_J[J_PosStartApproccioPrelLastra].Velocita			:= J_Par.Vel_Vuoto;
Programma_J[J_PosStartApproccioPrelLastra].Accelerazione		:= J_Par.Acc_Vuoto;
Programma_J[J_PosStartApproccioPrelLastra].Decelerazione		:= J_Par.Dec_Vuoto;
Programma_J[J_PosStartApproccioPrelLastra].Jerk				:= J_Par.Jerk_Vuoto;
Programma_J[J_PosStartApproccioPrelLastra].DisabilitaTasteggio	:= TRUE;

(* Programma 14 Asse J : Rotazione a quota di START APPROCCIO per prelievo su cavallina *)
Programma_J[J_PosSfogliatura].ID 					:= INT_TO_UINT(J_PosSfogliatura);
Programma_J[J_PosSfogliatura].Quota_Destinazione	:= Quota_Rotazione_Sfogliatura;
Programma_J[J_PosSfogliatura].Velocita			:= J_Par.Vel_Ridotta;
Programma_J[J_PosSfogliatura].Accelerazione		:= J_Par.Acc_Carico;
Programma_J[J_PosSfogliatura].Decelerazione		:= J_Par.Dec_Carico;
Programma_J[J_PosSfogliatura].Jerk				:= J_Par.Jerk_Carico;
//Programma_J[J_PosSfogliatura].DisabilitaTasteggio	:= FALSE;
Programma_J[J_PosSfogliatura].DisabilitaTasteggio	:= TRUE; //24-7-2025

(* Programma 17 Asse J : Posizione di PosPostScarico in deposito *)
Programma_J[J_PosPostScarico].ID 					:= INT_TO_UINT(J_PosPostScarico);
Programma_J[J_PosPostScarico].Quota_Destinazione	:= Quota_PostScaricoJ;
Programma_J[J_PosPostScarico].Velocita			:= J_Par.Vel_Vuoto;
Programma_J[J_PosPostScarico].Accelerazione		:= J_Par.Acc_Carico;
Programma_J[J_PosPostScarico].Decelerazione		:= J_Par.Dec_Carico;
Programma_J[J_PosPostScarico].Jerk				:= J_Par.Jerk_Carico;
Programma_J[J_PosPostScarico].DisabilitaTasteggio	:= TRUE;

(* Programma 18 Asse J : Traslazione a quota di FUORI INGOMBRO Pos Acrual*)
Programma_J[J_PosFuoriIngombroPosAttuale].ID 					:= INT_TO_UINT(J_PosFuoriIngombroPosAttuale);
Programma_J[J_PosFuoriIngombroPosAttuale].Quota_Destinazione	:= Quota_Fuori_Ingombro_AttualeJ;
Programma_J[J_PosFuoriIngombroPosAttuale].Velocita				:= J_Par.Vel_Vuoto;
Programma_J[J_PosFuoriIngombroPosAttuale].Accelerazione			:= J_Par.Acc_Vuoto;
Programma_J[J_PosFuoriIngombroPosAttuale].Decelerazione			:= J_Par.Dec_Vuoto;
Programma_J[J_PosFuoriIngombroPosAttuale].Jerk					:= J_Par.Jerk_Vuoto;
Programma_J[J_PosFuoriIngombroPosAttuale].DisabilitaTasteggio	:= TRUE;


(* Programma 0 Asse J : Traslazione a quota di 0 Grados) *)
Programma_J[Pos0TrasporteCavallete].ID 						:= Pos0TrasporteCavallete;
Programma_J[Pos0TrasporteCavallete].Quota_Destinazione		:= Pos0TrasporteCavallete;
Programma_J[Pos0TrasporteCavallete].Velocita				:= J_Par.Vel_Vuoto;
Programma_J[Pos0TrasporteCavallete].Accelerazione			:= J_Par.Acc_Vuoto;
Programma_J[Pos0TrasporteCavallete].Decelerazione			:= J_Par.Dec_Vuoto;
Programma_J[Pos0TrasporteCavallete].Jerk					:= J_Par.Jerk_Vuoto;
Programma_J[Pos0TrasporteCavallete].DisabilitaTasteggio	:= TRUE;


(* Programma 180 Asse J : Traslazione a quota di 180 Grados) *)
Programma_J[Pos180TrasporteCavallete].ID 						:= Pos180TrasporteCavallete;
Programma_J[Pos180TrasporteCavallete].Quota_Destinazione		:= Pos180TrasporteCavallete;
Programma_J[Pos180TrasporteCavallete].Velocita					:= J_Par.Vel_Vuoto;
Programma_J[Pos180TrasporteCavallete].Accelerazione				:= J_Par.Acc_Vuoto;
Programma_J[Pos180TrasporteCavallete].Decelerazione				:= J_Par.Dec_Vuoto;
Programma_J[Pos180TrasporteCavallete].Jerk						:= J_Par.Jerk_Vuoto;
Programma_J[Pos180TrasporteCavallete].DisabilitaTasteggio		:= TRUE;


Inizializzato := TRUE;

END_FUNCTION_BLOCK

// ---- POUs/TFCicliDiLavoro/Lastre/TFCiclo_Di_Riposo_Lastre.TcPOU
FUNCTION_BLOCK TFCiclo_Di_Riposo_Lastre
VAR_INPUT
	Ciclo 		: POINTER TO Stato_Ciclo_Lavoro;
	Programma  : POINTER TO TFProgramma_Ciclo_Riposo_Lastre;
	ModuleAX_X : POINTER TO TFModulePalletizer_Ax;
	ModuleAX_Y : POINTER TO TFModulePalletizer_Ax;
	ModuleAX_Z : POINTER TO TFModulePalletizer_Ax;
	ModuleAX_J : POINTER TO TFModulePalletizer_AxJ_Lastre;
	StartInterpolazioneAssi : POINTER TO BOOL;
	ModulePinza : POINTER TO TFModulePalletizer_Pinza;
	QuotaPassModePuntoIntermedio : ARRAY [1..3] OF REAL;
	AbilitazioneGlobalePassMode	: BOOL;
	InterrompiCiclo : BOOL;
	Abilita_Ciclo_Step : BOOL;
	Command_Step : BOOL;
	AbilitazioneAnticipoDinamicoMovimenti : BOOL;
END_VAR
VAR_OUTPUT
	STEPDone	: BOOL;
	Errore : uint;
END_VAR
VAR
	StepInto : BOOL;
	PinzaVerticale				: BOOL;
END_VAR

(* Set della variabile che mi permette di fare lo STEP nel ciclo *)
StepInto := (Abilita_Ciclo_Step AND Command_Step) OR NOT Abilita_Ciclo_Step;

(* Reset Anticipo Dinamico se non ho l'abilitazione *)
IF NOT AbilitazioneAnticipoDinamicoMovimenti  OR NOT HMI_DisabilitaAnticipiGLOBALE THEN
	QuotaAnticipoDinamicaX_Raggiunta := FALSE;
	QuotaAnticipoDinamicaY_Raggiunta := FALSE;
	QuotaAnticipoDinamicaZ_Raggiunta := FALSE;
	QuotaAnticipoDinamicaJ_Raggiunta := FALSE;
END_IF

PinzaVerticale := ModuleAX_J^.Ax^.Status.ActPosition > 95 OR ModuleAX_J^.Ax^.Status.ActPosition < 85;

IF NOT InterrompiCiclo THEN
	IF Ciclo^.Stato = TERMINATO OR Ciclo^.Stato = ANNULLATO OR Ciclo^.Stato = INTERROTTO THEN
		 Ciclo^.Passo := 0;
	END_IF
	 Ciclo^.Stato := IN_ESECUZIONE;
	CASE  Ciclo^.Passo OF
	(* Case 0 *)
			0:   Ciclo^.Stato := IN_ESECUZIONE;
				 Ciclo^.Passo := 10;
				 Programma_Z[Z_PosFuoriIngombroRiposo].Stato 			:= NON_ESEGUITO;
				 Programma_Y[Y_PosFuoriIngombroRiposo].Stato			:= NON_ESEGUITO;
				 Programma_J[J_PosFuoriIngombro].Stato					:= NON_ESEGUITO;
				 Programma_X[X_PosDiRiposo].Stato 						:= NON_ESEGUITO;
				 Programma_Z[Z_PosDiRiposo].Stato						:= NON_ESEGUITO;
				 Programma_J[J_PosDiRiposo].Stato						:= NON_ESEGUITO;
				 
				 ProgrammaToModule_X.Stato := NON_ESEGUITO;
				 ProgrammaToModule_Y.Stato := NON_ESEGUITO;
				 ProgrammaToModule_Z.Stato := NON_ESEGUITO;
				 ProgrammaToModule_J.Stato := NON_ESEGUITO;

				 STEPDone := FALSE;
		
			(* Case 10 - Spengo aspirazione *)
			10:	IF ModulePinza^.CmdNext.Code = '' THEN
					TFParametersArrayClear(ADR(ParametersArray));
					TFCommandSend(CmdUNLOAD,ParametersArray,ModulePinza^.Cmd);
					ModulePinza^.IN.RichiestaRicalibrazioneOvemEsterna := TRUE; //Ricalibrazione automatica OVEM
					Ciclo^.Passo := 11;
				END_IF
				
			11: IF TFStateCodeGet(ModulePinza^.State) = StateUNLOAD_END THEN
					Ciclo^.Passo := 20;
				END_IF		
				
			(* Case 20 - PROGRAMMA[0] ASSE Z -> TRASLAZIONE A QUOTA DI FUORI INGOMBRO *)	
			(*
			19:	 Ciclo^.Stato := IN_ESECUZIONE;
				IF StepInto THEN
					Programma_Z[Z_PosFuoriIngombroRiposo].Stato 			:= DA_ESEGUIRE;
					Programma_Z[Z_PosFuoriIngombroRiposo].InterpolaAsse 	:= NO_INTERPOLAZIONE_ASSE;
					ProgrammaToModule_Z 									:= Programma_Z[Z_PosFuoriIngombroRiposo];
					Ciclo^.Passo := 20;
					STEPDone := FALSE;
				END_IF
				*)
			(* Case 20 - PROGRAMMA[106] ASSE Z -> TRASLAZIONE A QUOTA DI FUORI INGOMBRO *)	
			20:	
				IF StepInto THEN
					IF PinzaVerticale AND NOT AsseXInFinestraDiPrelievo THEN
						Programma_Z[Z_PosFuoriIngombroRiposo].Stato 			:= DA_ESEGUIRE;
						//Programma_Z[Z_PosFuoriIngombroRiposo].InterpolaAsse 	:= INTERPOLAZIONE_ASSE (* INTERPOLAZIONE_ASSE*);
						Programma_Z[Z_PosFuoriIngombroRiposo].InterpolaAsse 	:= No_INTERPOLAZIONE_ASSE (* INTERPOLAZIONE_ASSE*);
						ProgrammaToModule_Z 									:= Programma_Z[Z_PosFuoriIngombroRiposo];

						Programma_Y[Y_PosFuoriIngombroRiposo].Stato 			:= DA_ESEGUIRE;
						Programma_Y[Y_PosFuoriIngombroRiposo].InterpolaAsse 	:= INTERPOLAZIONE_ASSE (* INTERPOLAZIONE_ASSE*);
						ProgrammaToModule_Y 										:= Programma_Y[Y_PosFuoriIngombroRiposo];

						Programma_J[J_PosFuoriIngombro].Stato 			:= DA_ESEGUIRE;
						Programma_J[J_PosFuoriIngombro].InterpolaAsse 	:= INTERPOLAZIONE_ASSE (* INTERPOLAZIONE_ASSE*);
						ProgrammaToModule_J 							:= Programma_J[J_PosFuoriIngombro];

						StartInterpolazioneAssi^ 	:= TRUE; //Abilito l'interpolazione degli assi
					ELSE
						Programma_Z[Z_PosFuoriIngombroRiposo].Stato 			:= DA_ESEGUIRE;
						//Programma_Z[Z_PosFuoriIngombroRiposo].InterpolaAsse 	:= INTERPOLAZIONE_ASSE;
						Programma_Z[Z_PosFuoriIngombroRiposo].InterpolaAsse 	:= No_INTERPOLAZIONE_ASSE;
						ProgrammaToModule_Z 									:= Programma_Z[Z_PosFuoriIngombroRiposo];
					END_IF
					Ciclo^.Passo := 21;
					STEPDone := FALSE;
				END_IF
				
			(* Case 21 - Attesa completamento del comando MOVETOPOS o del raggiungimento quota di Pre-Movimento se abilitata la funzione*)
			21: IF (Programma_Z[Z_PosFuoriIngombroRiposo].Stato = TERMINATO OR
					Asse_Z_InFinestraDiPassMode OR 
					QuotaAnticipoDinamicaZ_Raggiunta)  AND 
					((PinzaVerticale AND NOT AsseXInFinestraDiPrelievo AND 
					(Programma_Y[Y_PosFuoriIngombroRiposo].Stato = TERMINATO OR 
					Asse_Y_InFinestraDiPassMode) AND 
					(Programma_J[J_PosFuoriIngombro].Stato = TERMINATO OR 
					Asse_J_InFinestraDiPassMode)) OR NOT PinzaVerticale OR AsseXInFinestraDiPrelievo) THEN
						Ciclo^.Passo := 24;
						STEPDone := TRUE;
				ELSIF Programma_Z[Z_PosFuoriIngombroRiposo].Stato = INTERROTTO THEN
					Ciclo^.Passo := 21;										
				END_IF
				
		(*	22: IF Programma_Z[Z_PosFuoriIngombroRiposo].Stato = INTERROTTO THEN
					 Ciclo^.Passo := 22;
				ELSIF Programma_Z[Z_PosFuoriIngombroRiposo].Stato = TERMINATO OR 
						Asse_Z_InFinestraDiPassMode OR 
						QuotaAnticipoDinamicaZ_Raggiunta THEN
							IF StepInto THEN
								Programma_J[J_PosFuoriIngombro].Stato 			:= DA_ESEGUIRE;
								Programma_J[J_PosFuoriIngombro].InterpolaAsse 	:= NO_INTERPOLAZIONE_ASSE;
								ProgrammaToModule_J		 						:= Programma_J[J_PosFuoriIngombro];
								Ciclo^.Passo := 23;
								STEPDone := FALSE;
							END_IF									
				END_IF		
			23: IF Programma_Z[Z_PosFuoriIngombroRiposo].Stato = INTERROTTO OR 
					Programma_J[J_PosFuoriIngombro].Stato = INTERROTTO THEN
					 Ciclo^.Passo := 23;
				ELSIF (Programma_Z[Z_PosFuoriIngombroRiposo].Stato = TERMINATO) AND// OR Asse_Z_InFinestraDiPassMode OR QuotaAnticipoDinamicaZ_Raggiunta) AND 
					(Programma_J[J_PosFuoriIngombro].Stato = TERMINATO OR Asse_J_InFinestraDiPassMode OR QuotaAnticipoDinamicaJ_Raggiunta) THEN
						Ciclo^.Passo := 24;
						STEPDone := TRUE;										
				END_IF	
							
				
			(* Case 24 - Scelgo in quale direzione devo muovermi per primo a seconda della disposizione delle postazioni *)	
			24:	
				CASE ASSE_DISPOSIZIONE_POSTAZIONI OF
					
					LUNGO_X:
							Ciclo^.Passo := 25;
				
					LUNGO_Y:	
							Ciclo^.Passo := 50;
			
				END_CASE
				
			(* Case 25 - Vado a quota di fuori ingombro con Y *)
			25:	IF Programma_Z[Z_PosFuoriIngombroRiposo].Stato = INTERROTTO OR
					Programma_J[J_PosFuoriIngombro].Stato = INTERROTTO THEN
						Ciclo^.Passo := 25;										
				ELSE
					IF StepInto THEN
						Programma_Y[Y_PosFuoriIngombroRiposo].Stato 			:= DA_ESEGUIRE;
						Programma_Y[Y_PosFuoriIngombroRiposo].InterpolaAsse 	:= NO_INTERPOLAZIONE_ASSE;
						ProgrammaToModule_Y 									:= Programma_Y[Y_PosFuoriIngombroRiposo];
						Ciclo^.Passo := 26;
						STEPDone := FALSE;
					END_IF
				END_IF*)

	
			(* Case 24 - Vado a quota di fuori ingombro y e j  *)
			24:
				IF Programma_Z[Z_PosFuoriIngombroRiposo].Stato = INTERROTTO OR 
					((PinzaVerticale AND NOT AsseXInFinestraDiPrelievo)AND(Programma_Y[Y_PosFuoriIngombroRiposo].Stato = INTERROTTO OR
					Programma_J[J_PosFuoriIngombro].Stato = INTERROTTO)) THEN
						Ciclo^.Passo := 24;										
				ELSE
					IF StepInto THEN
						IF (NOT PinzaVerticale AND NOT AsseXInFinestraDiPrelievo) THEN
							Programma_Y[Y_PosFuoriIngombroRiposo].Stato 			:= DA_ESEGUIRE;
							Programma_Y[Y_PosFuoriIngombroRiposo].InterpolaAsse 	:= INTERPOLAZIONE_ASSE;
							ProgrammaToModule_Y 										:= Programma_Y[Y_PosFuoriIngombroRiposo];
	
							Programma_J[J_PosFuoriIngombro].Stato 			:= DA_ESEGUIRE;
							Programma_J[J_PosFuoriIngombro].InterpolaAsse 	:= INTERPOLAZIONE_ASSE;
							ProgrammaToModule_J 							:= Programma_J[J_PosFuoriIngombro];
						END_IF
						IF NOT FuoriIngombroYNecessario THEN
							Programma_X[X_PosDiRiposo].Stato 			:= DA_ESEGUIRE;
							Programma_X[X_PosDiRiposo].InterpolaAsse 	:= INTERPOLAZIONE_ASSE;
							ProgrammaToModule_X 										:= Programma_X[X_PosDiRiposo];
							Ciclo^.Passo := 31;
						ELSE
							Ciclo^.Passo := 25;
						END_IF
						StartInterpolazioneAssi^ 	:= TRUE; //Abilito l'interpolazione degli assi
						STEPDone 					:= FALSE;
					END_IF
				END_IF
				
			(* Case 25 - *)
			25: IF Programma_Z[Z_PosFuoriIngombroRiposo].Stato = INTERROTTO OR  
					(Programma_X[X_PosDiRiposo].Stato = INTERROTTO AND NOT FuoriIngombroYNecessario) OR
					Programma_Y[Y_PosFuoriIngombroRiposo].Stato = INTERROTTO OR
					Programma_J[J_PosFuoriIngombro].Stato = INTERROTTO THEN
						Ciclo^.Passo := 25;
				ELSIF (Programma_Y[Y_PosFuoriIngombroRiposo].Stato = TERMINATO OR 
					Asse_Y_InFinestraDiPassMode) AND 
					(Programma_J[J_PosFuoriIngombro].Stato = TERMINATO OR 
					Asse_J_InFinestraDiPassMode) THEN	
						Ciclo^.Passo := 30;
						STEPDone := TRUE;									
				END_IF
					
			(* Case 26 - Check se a quota di fuori ingombro con Y *)		
			26:	IF Programma_Y[Y_PosFuoriIngombroRiposo].Stato = INTERROTTO OR 
					Programma_Z[Z_PosFuoriIngombroRiposo].Stato = INTERROTTO OR 
					Programma_J[J_PosFuoriIngombro].Stato = INTERROTTO THEN
						Ciclo^.Passo := 26;
				ELSE	
					IF Programma_Y[Y_PosFuoriIngombroRiposo].Stato = TERMINATO OR 
						Asse_Y_InFinestraDiPassMode THEN
							Ciclo^.Passo := 30;
							STEPDone := TRUE;							
					END_IF
				END_IF
										
			(* Case 30 - PROGRAMMA[0] ASSE X  -> TRASLAZIONE A QUOTA DI RIPOSO  *)	
			30:	IF Programma_Z[Z_PosFuoriIngombroRiposo].Stato = INTERROTTO OR 
					Programma_Y[Y_PosFuoriIngombroRiposo].Stato = INTERROTTO OR 
					Programma_J[J_PosFuoriIngombro].Stato = INTERROTTO THEN
						Ciclo^.Passo := 30;										
				ELSE
					IF StepInto THEN
						Programma_X[X_PosDiRiposo].Stato := DA_ESEGUIRE;
						Programma_X[X_PosDiRiposo].InterpolaAsse := NO_INTERPOLAZIONE_ASSE;
						ProgrammaToModule_X := Programma_X[X_PosDiRiposo];
					
						Ciclo^.Passo := 31;
						STEPDone := FALSE;
					END_IF
				END_IF			
				
			(* Case 31 -  Attesa completamento del comando MOVETOPOS o del raggiungimento quota di Pre-Movimento se abilitata la funzione *)
			31: 
				IF Programma_X[X_PosDiRiposo].Stato = INTERROTTO OR
					Programma_Y[Y_PosFuoriIngombroRiposo].Stato = INTERROTTO OR
					Programma_Z[Z_PosFuoriIngombroRiposo].Stato = INTERROTTO OR 
					Programma_J[J_PosFuoriIngombro].Stato = INTERROTTO THEN
						Ciclo^.Passo := 31;
				ELSE	
					IF (Programma_X[X_PosDiRiposo].Stato = TERMINATO OR Asse_X_InFinestraDiPassMode OR QuotaAnticipoDinamicaX_Raggiunta) THEN 
						Ciclo^.Passo := 32;
						STEPDone := TRUE;							
					END_IF
				END_IF
				
			(* Case 32 - Vado a quota di riposo con Y,Z,J *)
			32:
				IF Programma_X[X_PosDiRiposo].Stato = INTERROTTO OR
					Programma_Y[Y_PosFuoriIngombroRiposo].Stato = INTERROTTO OR
					Programma_Z[Z_PosFuoriIngombroRiposo].Stato = INTERROTTO OR 
					Programma_J[J_PosFuoriIngombro].Stato = INTERROTTO THEN
						Ciclo^.Passo := 32;										
				ELSE
					IF StepInto THEN
						TFParametersArrayClear(ADR(ParametersArray));
						Programma_Y[Y_PosDiRiposo].Stato := DA_ESEGUIRE;
						Programma_Y[Y_PosDiRiposo].InterpolaAsse := INTERPOLAZIONE_ASSE;
					
						Programma_Z[Z_PosDiRiposo].Stato := DA_ESEGUIRE;
						//Programma_Z[Z_PosDiRiposo].InterpolaAsse := INTERPOLAZIONE_ASSE;
						Programma_Z[Z_PosDiRiposo].InterpolaAsse := NO_INTERPOLAZIONE_ASSE;
						
						Programma_J[J_PosDiRiposo].Stato := DA_ESEGUIRE;
						Programma_J[J_PosDiRiposo].InterpolaAsse := INTERPOLAZIONE_ASSE;
						
						ProgrammaToModule_Y := Programma_Y[Y_PosDiRiposo];
						ProgrammaToModule_Z := Programma_Z[Z_PosDiRiposo];
						ProgrammaToModule_J := Programma_J[J_PosDiRiposo];
						
						StartInterpolazioneAssi^ := TRUE; //Abilito l'interpolazione degli assi
												
						Ciclo^.Passo := 90;
						STEPDone := FALSE;
					END_IF
				END_IF
												
			(* Case 50 - Vado a quota di RIPOSO con X *)
			50:	IF Programma_Z[Z_PosFuoriIngombroRiposo].Stato = INTERROTTO OR
					Programma_J[J_PosFuoriIngombro].Stato = INTERROTTO THEN
						Ciclo^.Passo := 50;										
				ELSE
					IF StepInto THEN
						Programma_X[X_PosDiRiposo].Stato 				:= DA_ESEGUIRE;
						Programma_X[X_PosDiRiposo].InterpolaAsse 		:= NO_INTERPOLAZIONE_ASSE;
						ProgrammaToModule_X 							:= Programma_X[X_PosDiRiposo];
						Ciclo^.Passo := 51;
						STEPDone := FALSE;
					END_IF
				END_IF
					
			(* Case 51 - Check se a quota di fuori RIPOSO con X *)		
			51:	IF Programma_X[X_PosDiRiposo].Stato = INTERROTTO OR 
					Programma_Z[Z_PosFuoriIngombroRiposo].Stato = INTERROTTO OR 
					Programma_J[J_PosFuoriIngombro].Stato = INTERROTTO THEN
						Ciclo^.Passo := 51;
				ELSE	
					IF Programma_X[X_PosDiRiposo].Stato = TERMINATO OR Asse_X_InFinestraDiPassMode OR QuotaAnticipoDinamicaX_Raggiunta THEN
						Ciclo^.Passo := 52;
						STEPDone := TRUE;							
					END_IF
				END_IF
												
			(* Case 52 - Vado a quota di riposo con Y,Z,J *)
			52:
				IF Programma_X[X_PosDiRiposo].Stato = INTERROTTO OR
					Programma_Z[Z_PosFuoriIngombroRiposo].Stato = INTERROTTO OR 
					Programma_J[J_PosFuoriIngombro].Stato = INTERROTTO THEN
						Ciclo^.Passo := 52;										
				ELSE
					IF StepInto THEN
						TFParametersArrayClear(ADR(ParametersArray));
						Programma_Y[Y_PosDiRiposo].Stato 			:= DA_ESEGUIRE;
						Programma_Y[Y_PosDiRiposo].InterpolaAsse 	:= INTERPOLAZIONE_ASSE;
					
						//Programma_Z[Z_PosDiRiposo].Stato 			:= DA_ESEGUIRE;
						//Programma_Z[Z_PosDiRiposo].InterpolaAsse 	:= INTERPOLAZIONE_ASSE;
						
						Programma_J[J_PosDiRiposo].Stato 			:= DA_ESEGUIRE;
						Programma_J[J_PosDiRiposo].InterpolaAsse 	:= INTERPOLAZIONE_ASSE;
						
						ProgrammaToModule_Y := Programma_Y[Y_PosDiRiposo];
						//ProgrammaToModule_Z := Programma_Z[Z_PosDiRiposo];
						ProgrammaToModule_J := Programma_J[J_PosDiRiposo];
						
						StartInterpolazioneAssi^ := TRUE; //Abilito l'interpolazione degli assi
												
						Ciclo^.Passo := 53;
						STEPDone := FALSE;
					END_IF
				END_IF

			(* Case 53 - Vado a quota di riposo con Z *)
			53:
				IF Programma_X[X_PosDiRiposo].Stato = INTERROTTO OR
					Programma_Y[Y_PosDiRiposo].Stato = INTERROTTO OR 
					Programma_J[J_PosDiRiposo].Stato = INTERROTTO THEN
						Ciclo^.Passo := 53;										
				ELSE
					IF StepInto THEN
						IF Programma_Y[Y_PosDiRiposo].Stato = TERMINATO (*OR Asse_Y_InFinestraDiPassMode)*) AND 
							Programma_J[J_PosDiRiposo].Stato = TERMINATO (*OR Asse_J_InFinestraDiPassMode)*) THEN
					
								Programma_Z[Z_PosDiRiposo].Stato 			:= DA_ESEGUIRE;
								Programma_Z[Z_PosDiRiposo].InterpolaAsse 	:= NO_INTERPOLAZIONE_ASSE;
								
								ProgrammaToModule_Z := Programma_Z[Z_PosDiRiposo];
								
								StartInterpolazioneAssi^ := FALSE; //Abilito l'interpolazione degli assi
														
								Ciclo^.Passo := 90;
								STEPDone := FALSE;
						END_IF
					END_IF
				END_IF

			(* Case 90 - Attesa completamento posizionamento di tutti gli assi *)
			90: 
				IF Programma_Y[Y_PosDiRiposo].Stato = TERMINATO (*OR Asse_Y_InFinestraDiPassMode)*) AND 
					Programma_J[J_PosDiRiposo].Stato = TERMINATO (*OR Asse_J_InFinestraDiPassMode)*) AND
					Programma_X[X_PosDiRiposo].Stato = TERMINATO (*OR Asse_X_InFinestraDiPassMode)*) AND 
					Programma_Z[Z_PosDiRiposo].Stato = TERMINATO (*OR Asse_Z_InFinestraDiPassMode)*) THEN
						Ciclo^.Passo := 1000;
						STEPDone := TRUE;
				ELSIF Programma_Y[Y_PosDiRiposo].Stato = INTERROTTO OR 
					Programma_J[J_PosDiRiposo].Stato = INTERROTTO OR 
					Programma_X[X_PosDiRiposo].Stato = INTERROTTO OR
					Programma_Z[Z_PosDiRiposo].Stato = TERMINATO THEN

						Ciclo^.Passo := 90;									
				END_IF
				
			(* Case 1000 *)
			1000:
				 Ciclo^.Stato := TERMINATO;
				 Ciclo^.Passo := 1000;
	ELSE;
	END_CASE;
ELSE								//Se il ciclo deve essere interrotto, setto il suo nuovo stato
	 Ciclo^.Stato := INTERROTTO;
END_IF

END_FUNCTION_BLOCK

// ---- POUs/TFCicliDiLavoro/Lastre/Cicli di Prelievo Lastre/TFCiclo_Prelievo_Falda.TcPOU
FUNCTION_BLOCK TFCiclo_Prelievo_Falda
VAR_INPUT
	Ciclo 		: POINTER TO Stato_Ciclo_Lavoro;
	Programma  : POINTER TO TFProgramma_Ciclo_Falda_Lastre;
	ModuleAX_X : POINTER TO TFModulePalletizer_Ax;
	ModuleAX_Y : POINTER TO TFModulePalletizer_Ax;
	ModuleAX_Z : POINTER TO TFModulePalletizer_Ax;
	ModuleAX_J : POINTER TO TFModulePalletizer_AxJ_Lastre;
	StartInterpolazioneAssi : POINTER TO BOOL;
	QuotaPassModePuntoIntermedio : ARRAY [1..3] OF REAL;
	ModulePinza : POINTER TO TFModulePalletizer_Pinza;
	AbilitazioneGlobalePassMode	: BOOL;
	InterrompiCiclo : BOOL;
	Abilita_Ciclo_Step : BOOL;
	Command_Step : BOOL;
	AbilitazioneAnticipoDinamicoMovimenti : bool;
END_VAR
VAR_OUTPUT
	STEPDone	: BOOL;
END_VAR
VAR
	ComandoInviatoTRIG : bool;
	StepInto: BOOL;
END_VAR

(* Set della variabile che mi permette di fare lo STEP nel ciclo *)
StepInto := (Abilita_Ciclo_Step AND Command_Step) OR NOT Abilita_Ciclo_Step;

(* Reset Anticipo Dinamico se non ho l'abilitazione *)
IF NOT AbilitazioneAnticipoDinamicoMovimenti  OR NOT HMI_DisabilitaAnticipiGLOBALE THEN
	QuotaAnticipoDinamicaX_Raggiunta := FALSE;
	QuotaAnticipoDinamicaY_Raggiunta := FALSE;
	QuotaAnticipoDinamicaZ_Raggiunta := FALSE;
END_IF

IF NOT InterrompiCiclo THEN
	IF Ciclo^.Stato = TERMINATO OR Ciclo^.Stato = ANNULLATO THEN
		Ciclo^.Passo := 0;
	ELSIF Ciclo^.Stato = INTERROTTO THEN
		Ciclo^.Passo := 999;
	END_IF
	Ciclo^.Stato := IN_ESECUZIONE;
	CASE Ciclo^.Passo OF
	(* Case 0 *)
			0:  Ciclo^.Stato := IN_ESECUZIONE;
				Ciclo^.Passo := 10;
				STEPDone := FALSE;
		
			(* Case 10 - Spengo aspirazione *)
			10:	IF ModulePinza^.CmdNext.Code = '' THEN
					IF (Abilita_Ciclo_Step AND Command_Step) OR NOT Abilita_Ciclo_Step THEN
						TFParametersArrayClear(ADR(ParametersArray));
						TFCommandSend(CmdUNLOAD,ParametersArray,ModulePinza^.Cmd);
						Ciclo^.Passo := 11;
						STEPDone := FALSE;
					END_IF
				END_IF
			(* Case 11 - Attesa aspirazione off*)
			11:
				IF TFStateCodeGet(ModulePinza^.State) = StateERROR  THEN
					Ciclo^.Passo := 0;	
					STEPDone := TRUE;
				ELSIF NOT TFStateCodeGet(ModulePinza^.State) = StateUNLOAD_RUN  THEN
					Ciclo^.Passo := 10;	
					STEPDone := TRUE;								
				ELSE
					IF TFStateCodeGet(ModulePinza^.State) = StateUNLOAD_END THEN
						Ciclo^.Passo := 20;
						STEPDone := TRUE;
					END_IF	
				END_IF;
				
			(* Case 20 - PROGRAMMA[0] ASSE Z -> TRASLAZIONE A QUOTA DI FUORI INGOMBRO *)	
			20:	Ciclo^.Stato := IN_ESECUZIONE;
				IF StepInto THEN
					TFParametersArrayClear(ADR(ParametersArray));
					Programma_Z[54].Stato := DA_ESEGUIRE;
					Programma_Z[54].InterpolaAsse := NO_INTERPOLAZIONE_ASSE;//FALSE;//NO_INTERPOLAZIONE_ASSE
					ProgrammaToModule_Z := Programma_Z[54];
					Ciclo^.Passo := 21;
					STEPDone := FALSE;
				END_IF
				
			(* Case 21 - Attesa completamento del comando MOVETOPOS o del raggiungimento quota di Pre-Movimento se abilitata la funzione*)
			21: 
				IF Programma_Z[54].Stato = TERMINATO OR 
					Asse_Z_InFinestraDiPassMode OR 
					QuotaAnticipoDinamicaZ_Raggiunta OR
					(ModuleAX_Z^.Ax^.Status.ActPosition >= QuotaFuoriIngombro_Z_AVUOTO-5) THEN
						Ciclo^.Passo := 22;
						STEPDone := TRUE;
				ELSIF Programma_Z[0].Stato = INTERROTTO THEN
					Ciclo^.Passo := 21;										
				END_IF
				
			(* Case 22 - Attesa completamento del comando MOVETOPOS o del raggiungimento quota di Pre-Movimento se abilitata la funzione *)
			22: IF Programma_Z[54].Stato = INTERROTTO THEN
					Ciclo^.Passo := 20;
				ELSE	
					Ciclo^.Passo := 23;
					STEPDone := TRUE;									
				END_IF
				
			(* Case 23 - Vado a quota di fuori ingombro colonne con Y *)
			23:
				IF Programma_Z[54].Stato = INTERROTTO THEN
					 Ciclo^.Passo := 20;										
				ELSE
					//IF FuoriIngombroYNecessario THEN
						IF StepInto THEN
							TFParametersArrayClear(ADR(ParametersArray));
							Programma_Y[56].Stato := DA_ESEGUIRE;
							Programma_Y[56].InterpolaAsse := NO_INTERPOLAZIONE_ASSE;
							ProgrammaToModule_Y := Programma_Y[56];
							Ciclo^.Passo := 24;
							STEPDone := FALSE;
						END_IF
					//ELSE
					//	Ciclo^.Passo := 24;
					//	STEPDone := FALSE;
					//END_IF
				END_IF
			
			(* Case 24 - *)
			24: IF Programma_Z[54].Stato = INTERROTTO OR
					Programma_Y[56].Stato = INTERROTTO THEN
						Ciclo^.Passo := 20;
				ELSIF Programma_Y[56].Stato = TERMINATO OR Asse_Y_InFinestraDiPassMode THEN// OR NOT FuoriIngombroYNecessario THEN	
					Ciclo^.Passo := 40;
					STEPDone := TRUE;									
				END_IF
				
			(* Case 40 - PROGRAMMA[] ASSE Y -> TRASLAZIONE A QUOTA DI PRELIEVO FALDA  *)	
			40:	
				IF Programma_Z[54].Stato = INTERROTTO OR 
					Programma_Y[56].Stato = INTERROTTO THEN
						Ciclo_Pelievo_Falda.Passo := 20;										
				ELSE
					IF StepInto THEN
						TFParametersArrayClear(ADR(ParametersArray));
						
						Programma_X[51].Stato := DA_ESEGUIRE;
						(*IF NOT Pinza_InIngombroColonne_Destinazione THEN
							Programma_Y[51].Stato := DA_ESEGUIRE;
							Programma_Y[54].InterpolaAsse := INTERPOLAZIONE_ASSE;//TRUE;//NO_INTERPOLAZIONE_ASSE
							ProgrammaToModule_Y := Programma_Y[51];
						END_IF*)
						Programma_J[10].Stato := DA_ESEGUIRE;
						Programma_K[51].Stato := DA_ESEGUIRE;
						
						Programma_X[51].InterpolaAsse := INTERPOLAZIONE_ASSE;//TRUE;//NO_INTERPOLAZIONE_ASSE
						//Programma_Y[54].InterpolaAsse := INTERPOLAZIONE_ASSE;//TRUE;//NO_INTERPOLAZIONE_ASSE
						Programma_J[10].InterpolaAsse := INTERPOLAZIONE_ASSE;//TRUE;//NO_INTERPOLAZIONE_ASSE
						Programma_K[51].InterpolaAsse := NO_INTERPOLAZIONE_ASSE;//FALSE;//NO_INTERPOLAZIONE_ASSE
						
						ProgrammaToModule_X := Programma_X[51];
						//ProgrammaToModule_Y := Programma_Y[51];
						ProgrammaToModule_J := Programma_J[10];
						ProgrammaToModule_K := Programma_K[51];
						
						ProgrammaToModule_Z.InterpolaAsse := NO_INTERPOLAZIONE_ASSE;//FALSE;//NO_INTERPOLAZIONE_ASSE
						
						StartInterpolazioneAssi^ := TRUE; //Abilito l'interpolazione degli assi
						
						TFCommandSend(CmdLOAD,ParametersArray,ModulePinza^.Cmd);
						
						Ciclo^.Passo := 41;
						STEPDone := FALSE;
					END_IF
				END_IF
				
			(* Case 41 - PROGRAMMA[51] ASSE Y -> TRASLAZIONE A QUOTA DI PRELIEVO FALDA  *)	
			41:	
				IF Programma_Z[54].Stato = INTERROTTO OR 
					Programma_Y[56].Stato = INTERROTTO OR 
					Programma_J[10].Stato = INTERROTTO OR 
					Programma_K[51].Stato = INTERROTTO OR 
					Programma_X[51].Stato = INTERROTTO THEN
					  Ciclo_Pelievo_Falda.Passo := 20;										
				ELSE
					STEPDone := TRUE;
					IF QuotaX_ConsensoRotazionePinza_Raggiunta OR NOT Pinza_InIngombroColonne_Destinazione THEN 
						IF StepInto THEN
							TFParametersArrayClear(ADR(ParametersArray));
							Programma_Y[51].Stato := DA_ESEGUIRE;
							Programma_Y[51].InterpolaAsse := NO_INTERPOLAZIONE_ASSE;
							ProgrammaToModule_Y := Programma_Y[51];
							
							Ciclo^.Passo := 42;
							STEPDone := FALSE;
						END_IF
					END_IF
				END_IF
					
			(* Case 42 -  Attesa completamento del comando MOVETOPOS o del raggiungimento quota di Pre-Movimento se abilitata la funzione *)
			42: 
				ComandoInviatoTRIG := FALSE;
				IF Programma_Z[54].Stato = INTERROTTO OR 
					Programma_Y[51].Stato = INTERROTTO OR  
					Programma_J[10].Stato = INTERROTTO OR 
					Programma_K[51].Stato = INTERROTTO OR 
					Programma_X[51].Stato = INTERROTTO THEN
						Ciclo^.Passo := 20;	
				ELSIF (Programma_X[51].Stato = TERMINATO OR Asse_X_InFinestraDiPassMode OR QuotaAnticipoDinamicaX_Raggiunta) AND 
					(Programma_Y[51].Stato = TERMINATO OR Asse_Y_InFinestraDiPassMode) AND
					(Programma_J[10].Stato = TERMINATO OR Asse_J_InFinestraDiPassMode) THEN
						Ciclo^.Passo := 80;
						STEPDone := TRUE;							
				END_IF
							
			(* Case 80 - PROGRAMMA[51] ASSE Z -> TRASLAZIONE A QUOTA AMMESSA IN VELOCE DI PRELIEVO FALDA  *)
			80:
				IF Programma_X[51].Stato = INTERROTTO THEN
					Ciclo^.Passo := 40;		//NON DOVREBBE MAI CAPITARE IN QUESTO PUNTO								
				ELSE
					IF StepInto THEN
						TFParametersArrayClear(ADR(ParametersArray));
						Programma_Z[51].Stato := DA_ESEGUIRE;
						Programma_Z[51].InterpolaAsse := NO_INTERPOLAZIONE_ASSE;//FALSE;//NO_INTERPOLAZIONE_ASSE
						ProgrammaToModule_Z := Programma_Z[51];
						Ciclo^.Passo := 81;
						STEPDone := FALSE;
					END_IF
				END_IF
			(* Case 81 -  Attesa completamento del comando MOVETOPOS o del raggiungimento quota di Pre-Movimento se abilitata la funzione *)
			81: 
				IF Programma_X[51].Stato = INTERROTTO OR 
				Programma_Z[51].Stato = INTERROTTO THEN
					Ciclo^.Passo := 40;									
				ELSE
					IF (Programma_Z[51].Stato = TERMINATO OR
					(ModuleAX_Z^.Ax^.Status.ActPosition <= Programma^.Quota_StartLenta_Prelievo_Falda_Z + 50 AND Programma_Z[51].Stato = IN_ESECUZIONE)) AND
					Programma_X[51].Stato = TERMINATO THEN	// controllo che la X sia in posizione corretta per poter iniziare la lenta senza collisioni
						Ciclo^.Passo := 100;
						STEPDone := TRUE;
					END_IF	
				END_IF
			
		 	(* Case 100 - PROGRAMMA[52] ASSE Z -> TRASLAZIONE IN LENTA A QUOTA DI PRELIEVO FALDA  *)
			100:
				IF Programma_Z[51].Stato = INTERROTTO THEN
					Ciclo^.Passo := 40; //NON DOVREBBE ACCADERE										
				ELSE
					IF StepInto THEN
						Programma_Z[52].Stato := DA_ESEGUIRE;
						Programma_Z[52].InterpolaAsse := NO_INTERPOLAZIONE_ASSE;//FALSE;//NO_INTERPOLAZIONE_ASSE
						ProgrammaToModule_Z := Programma_Z[52];
						Ciclo^.Passo := 101;
						STEPDone := FALSE;
					END_IF
				END_IF
				
			(* Case 101 -  Attesa completamento del comando MOVETOPOS o del raggiungimento quota di Pre-Movimento se abilitata la funzione *)
			101: 
				IF Programma_Z[52].Stato = INTERROTTO THEN
					Ciclo^.Passo := 20; //NON DOVREBBE ACCADERE										
				ELSE
					IF Programma_Z[52].Stato = TERMINATO THEN
						Ciclo^.Passo := 1000;
						STEPDone := TRUE;
					END_IF	
				END_IF
				
				(* Case 1000 *)
			1000:
				Ciclo^.Stato := TERMINATO;
				Ciclo^.Passo := 1000;
				
			(* Case 9999 - Ciclo NON annullato o NON terminato*)
			9999:
				Ciclo^.Stato := INTERROTTO;
				Ciclo^.Passo := 9999;
	ELSE						
		;
			
	END_CASE;
ELSE								//Se il ciclo deve essere interrotto, setto il suo nuovo stato
	Ciclo^.Stato := INTERROTTO;
END_IF

END_FUNCTION_BLOCK

// ---- POUs/TFCicliDiLavoro/Lastre/Cicli di Deposito Lastre/TFCiclo_Deposito_Falda.TcPOU
FUNCTION_BLOCK TFCiclo_Deposito_Falda
VAR_INPUT
	Ciclo 		: POINTER TO Stato_Ciclo_Lavoro;
	Programma  : POINTER TO TFProgramma_Ciclo_Falda_Lastre;
	ModuleAX_X : POINTER TO TFModulePalletizer_Ax;
	ModuleAX_Y : POINTER TO TFModulePalletizer_Ax;
	ModuleAX_Z : POINTER TO TFModulePalletizer_Ax;
	ModuleAX_J : POINTER TO TFModulePalletizer_AxJ_Lastre;
	StartInterpolazioneAssi : POINTER TO BOOL;
	QuotaPassModePuntoIntermedio : ARRAY [1..3] OF REAL;
	ModulePinza : POINTER TO TFModulePalletizer_Pinza;
	TipoDiDeposito : UINT;
	AbilitazioneGlobalePassMode	: BOOL;
	InterrompiCiclo : BOOL;
	Abilita_Ciclo_Step : BOOL;
	Command_Step : BOOL;
	AbilitazioneAnticipoDinamicoMovimenti : BOOL;
END_VAR
VAR_OUTPUT
	STEPDone	: BOOL;
END_VAR
VAR
	StepInto: BOOL;
END_VAR

(* Set della variabile che mi permette di fare lo STEP nel ciclo *)
StepInto := (Abilita_Ciclo_Step AND Command_Step) OR NOT Abilita_Ciclo_Step;

(* Reset Anticipo Dinamico se non ho l'abilitazione *)
IF NOT AbilitazioneAnticipoDinamicoMovimenti  OR NOT HMI_DisabilitaAnticipiGLOBALE THEN
	QuotaAnticipoDinamicaX_Raggiunta := FALSE;
	QuotaAnticipoDinamicaY_Raggiunta := FALSE;
	QuotaAnticipoDinamicaZ_Raggiunta := FALSE;
END_IF

IF NOT InterrompiCiclo THEN
	IF Ciclo^.Stato = TERMINATO OR Ciclo^.Stato = ANNULLATO THEN
		Ciclo^.Passo := 0;
	ELSIF Ciclo^.Stato = INTERROTTO THEN
		Ciclo^.Passo := 999;
	END_IF
	Ciclo^.Stato := IN_ESECUZIONE;
	CASE Ciclo^.Passo OF
	(* Case 0 *)
			0:  Ciclo^.Stato := IN_ESECUZIONE;
				Ciclo^.Passo := 10;
				STEPDone := FALSE;
		
			(* Case 10 - PROGRAMMA[53] ASSE Z -> TRASLAZIONE A QUOTA DI "ATTESA CADUTA FALDA" *)	
			10:	
				Ciclo^.Stato := IN_ESECUZIONE;
				IF StepInto THEN
					Programma_Z[53].Stato := DA_ESEGUIRE;
					Programma_Z[53].InterpolaAsse := NO_INTERPOLAZIONE_ASSE;//FALSE;//NO_INTERPOLAZIONE_ASSE
					ProgrammaToModule_Z := Programma_Z[53];
					Ciclo^.Passo := 11;
					STEPDone := FALSE;
				END_IF
				
			(* Case 11 - Attesa completamento del comando MOVETOPOS o del raggiungimento quota di Pre-Movimento se abilitata la funzione*)
			11: 
				IF Programma_Z[53].Stato = TERMINATO OR
				(ModuleAX_Z^.Ax^.Status.ActPosition >= Programma^.Quota_Attesa_Caduta_Falda_Z - 50) THEN // con -30 faccio in modo che il programma successivo si innesti a quello in corso.. per non vedere lo stacco...
					Ciclo^.Passo := 20;
					STEPDone := TRUE;
				ELSIF Programma_Z[53].Stato = INTERROTTO THEN
					Ciclo^.Passo := 10;										
				END_IF
				
			(* Case 20 - PROGRAMMA[54] ASSE Z -> TRASLAZIONE A QUOTA DI FUORI INGOMBRO *)	
			20:	Ciclo^.Stato := IN_ESECUZIONE;
				IF StepInto THEN
					Programma_Z[54].Stato := DA_ESEGUIRE;
					Programma_Z[54].InterpolaAsse := NO_INTERPOLAZIONE_ASSE;//FALSE;//NO_INTERPOLAZIONE_ASSE
					ProgrammaToModule_Z := Programma_Z[54];
					Ciclo^.Passo := 21;
					STEPDone := FALSE;
				END_IF
				
			(* Case 21 - Attesa completamento del comando MOVETOPOS o del raggiungimento quota di Pre-Movimento se abilitata la funzione *)
			21: 
				IF Programma_Z[54].Stato = TERMINATO OR
					(ModuleAX_Z^.Ax^.Status.ActPosition >= QuotaFuoriIngombro_Z_ConFALDA) OR 
					(Asse_Z_InFinestraDiPassMode AND Programma_Z[54].Stato = IN_ESECUZIONE) THEN
						IF (TipoDiDeposito = DEPOSITO_FALDA_SU_CATASTA AND ((Mission.PPick-1)=Mission.PPlace)) THEN//Vado direttamente in prelievo senza fare il fuori ingombro SE devo depositare sulla catasta e la catasta è di fronte al mag. falde 
							Ciclo^.Passo := 40;
							STEPDone := TRUE;
						ELSE
							Ciclo^.Passo := 22;
							STEPDone := TRUE;
						END_IF
				ELSIF Programma_Z[54].Stato = INTERROTTO THEN
					Ciclo^.Passo := 20;										
				END_IF
				
			(* Case 22 - Vado a quota di fuori ingombro colonne con Y *)
			22:
				IF Programma_Z[54].Stato = INTERROTTO THEN
					 Ciclo^.Passo := 20;										
				ELSE
					IF StepInto THEN
						Programma_Y[66].Stato := DA_ESEGUIRE;
						Programma_Y[66].InterpolaAsse := NO_INTERPOLAZIONE_ASSE;
						ProgrammaToModule_Y := Programma_Y[66];
						Ciclo^.Passo := 23;
						STEPDone := FALSE;
					END_IF
				END_IF
					
			(* Case 23 - Arrivato a quota di fuori ingombro colonne con Y *)		
			23:
				IF Programma_Z[54].Stato = INTERROTTO OR 
					Programma_Y[66].Stato = INTERROTTO THEN
						Ciclo^.Passo := 20;
				ELSE	
					IF Programma_Y[66].Stato = TERMINATO OR Asse_Y_InFinestraDiPassMode THEN
						Ciclo^.Passo := 40;
						STEPDone := TRUE;							
					END_IF
				END_IF
				
			(* Case 40 - PROGRAMMA[..] ASSE  -> TRASLAZIONE A QUOTA DI DEPOSITO FALDA  *)	
			40:	
				IF Programma_Z[54].Stato = INTERROTTO THEN					
					Ciclo^.Passo := 20;										
				ELSE
					IF TipoDiDeposito = DEPOSITO_FALDA_SU_CATASTA THEN
						IF StepInto THEN
							Programma_X[52].Stato := DA_ESEGUIRE;
							Programma_X[52].InterpolaAsse := INTERPOLAZIONE_ASSE;//TRUE;//INTERPOLAZIONE_ASSE
							ProgrammaToModule_X := Programma_X[52];
							IF NOT Pinza_InIngombroColonne_Destinazione THEN
								Programma_Y[52].Stato := DA_ESEGUIRE;
								Programma_Y[52].InterpolaAsse := INTERPOLAZIONE_ASSE;//TRUE;//INTERPOLAZIONE_ASSE
								ProgrammaToModule_Y := Programma_Y[52];
							END_IF
							Programma_J[11].Stato := DA_ESEGUIRE;
							Programma_J[11].InterpolaAsse := INTERPOLAZIONE_ASSE;//TRUE;//INTERPOLAZIONE_ASSE
							ProgrammaToModule_J := Programma_J[11];
							
							Programma_K[53].Stato := DA_ESEGUIRE;
							Programma_K[53].InterpolaAsse := NO_INTERPOLAZIONE_ASSE;//FALSE;//NO_INTERPOLAZIONE_ASSE
							ProgrammaToModule_K := Programma_K[53];
							
							ProgrammaToModule_Z.InterpolaAsse := NO_INTERPOLAZIONE_ASSE;//FALSE;
							
							StartInterpolazioneAssi^ := TRUE; //Abilito l'interpolazione degli assi

							Ciclo^.Passo := 41;
							STEPDone := FALSE;
						END_IF
					ELSIF TipoDiDeposito = DEPOSITO_FALDA_SU_PIAZZOLA THEN
						IF StepInto THEN
							Programma_X[53].Stato := DA_ESEGUIRE;
							Programma_X[53].InterpolaAsse := INTERPOLAZIONE_ASSE;//TRUE;//INTERPOLAZIONE_ASSE
							ProgrammaToModule_X := Programma_X[53];
							(*IF NOT Pinza_InIngombroColonne_Destinazione THEN
								Programma_Y[53].Stato := DA_ESEGUIRE;
								Programma_Y[53].InterpolaAsse := INTERPOLAZIONE_ASSE;//TRUE;//INTERPOLAZIONE_ASSE
								ProgrammaToModule_Y := Programma_Y[53];
							END_IF*)
							Programma_J[11].Stato := DA_ESEGUIRE;
							Programma_J[11].InterpolaAsse := INTERPOLAZIONE_ASSE;//TRUE;//INTERPOLAZIONE_ASSE
							ProgrammaToModule_J := Programma_J[11];
							
							Programma_K[53].Stato := DA_ESEGUIRE;
							Programma_K[53].InterpolaAsse := NO_INTERPOLAZIONE_ASSE;//FALSE;//NO_INTERPOLAZIONE_ASSE
							ProgrammaToModule_K := Programma_K[53];
							
							StartInterpolazioneAssi^ := TRUE; //Abilito l'interpolazione degli assi							
						
							Ciclo^.Passo := 41;
							STEPDone := FALSE;
						END_IF
					ELSE
						;
					END_IF
				END_IF
			
			41: IF Programma_Z[54].Stato = INTERROTTO THEN					
					Ciclo^.Passo := 20;										
				ELSE
					STEPDone := TRUE;
					IF QuotaX_ConsensoRotazionePinza_Raggiunta OR NOT Pinza_InIngombroColonne_Destinazione THEN
						IF TipoDiDeposito = DEPOSITO_FALDA_SU_CATASTA THEN
							IF StepInto THEN
								Programma_Y[52].Stato := DA_ESEGUIRE;
								Programma_Y[52].InterpolaAsse := NO_INTERPOLAZIONE_ASSE;//TRUE;//INTERPOLAZIONE_ASSE
								ProgrammaToModule_Y := Programma_Y[52];
								
								Ciclo^.Passo := 42;
								STEPDone := FALSE;
							END_IF
						ELSIF TipoDiDeposito = DEPOSITO_FALDA_SU_PIAZZOLA THEN
							IF StepInto THEN
								Programma_Y[53].Stato := DA_ESEGUIRE;
								Programma_Y[53].InterpolaAsse := NO_INTERPOLAZIONE_ASSE;//TRUE;//INTERPOLAZIONE_ASSE
								ProgrammaToModule_Y := Programma_Y[53];
								
								Ciclo^.Passo := 42;
								STEPDone := FALSE;
							END_IF
						ELSE
							;
						END_IF
					END_IF
				END_IF	
						
			(* Case 42 -  Attesa completamento del comando MOVETOPOS o del raggiungimento quota di Pre-Movimento se abilitata la funzione *)
			42: 
				IF Programma_Z[54].Stato = INTERROTTO OR 
					(TipoDiDeposito = DEPOSITO_FALDA_SU_CATASTA AND Programma_X[52].Stato = INTERROTTO) OR 
					(TipoDiDeposito = DEPOSITO_FALDA_SU_PIAZZOLA AND Programma_X[53].Stato = INTERROTTO) OR
					(TipoDiDeposito = DEPOSITO_FALDA_SU_CATASTA  AND Programma_Y[52].Stato = INTERROTTO) OR
					(TipoDiDeposito = DEPOSITO_FALDA_SU_PIAZZOLA AND Programma_Y[53].Stato = INTERROTTO) OR
					Programma_J[11].Stato = INTERROTTO OR
					Programma_K[53].Stato = INTERROTTO THEN
						Ciclo^.Passo := 20;	
				(* Deposito su catasta *)
				ELSIF TipoDiDeposito = DEPOSITO_FALDA_SU_CATASTA THEN
					IF (Programma_X[52].Stato = TERMINATO OR Asse_X_InFinestraDiPassMode) AND
						(Programma_Y[52].Stato = TERMINATO OR Asse_Y_InFinestraDiPassMode) AND  
					  	Programma_J[11].Stato = TERMINATO AND 
						Programma_K[53].Stato = TERMINATO THEN 
							Ciclo^.Passo := 50;
							STEPDone := TRUE;
					END_IF
				(* Deposito Su piazzola *)
				ELSIF (Programma_X[53].Stato = TERMINATO OR Asse_X_InFinestraDiPassMode) AND 
					  (Programma_Y[53].Stato = TERMINATO OR Asse_Y_InFinestraDiPassMode) AND
					  Programma_J[11].Stato = TERMINATO AND
					  Programma_K[53].Stato = TERMINATO THEN 
							Ciclo^.Passo := 50;
							STEPDone := TRUE;								
				END_IF	
							
			(* Case 80 - PROGRAMMA[..] ASSE Z -> TRASLAZIONE A QUOTA AMMESSA IN VELOCE DI DEPOSITO FALDA  
			- DEPOSITO_FALDA_SU_CATASTA : PROGRAMMA[55] ASSE Z
			- DEPOSITO_FALDA_SU_PIAZZOLA : PROGRAMMA[57] ASSE Z *)
			50:
				IF TipoDiDeposito = DEPOSITO_FALDA_SU_CATASTA THEN
					IF StepInto THEN
						Programma_Z[55].Stato := DA_ESEGUIRE;
						Programma_Z[55].InterpolaAsse := NO_INTERPOLAZIONE_ASSE;//FALSE;//NO_INTERPOLAZIONE_ASSE
						ProgrammaToModule_Z := Programma_Z[55];
						Ciclo^.Passo := 52;
						STEPDone := FALSE;
					END_IF
				ELSIF TipoDiDeposito = DEPOSITO_FALDA_SU_PIAZZOLA THEN
					IF StepInto THEN
						Programma_Z[57].Stato := DA_ESEGUIRE;
						Programma_Z[57].InterpolaAsse := NO_INTERPOLAZIONE_ASSE;//FALSE;//NO_INTERPOLAZIONE_ASSE
						ProgrammaToModule_Z := Programma_Z[57];
						Ciclo^.Passo := 51;	//SALTO DIRETTAMENTE AL CASE 91 DOVE SI ASPETTA LA FINE DEL MOVIMENTO DELL'ASSE Z
						STEPDone := FALSE;
					END_IF
				ELSE
					;
				END_IF
					
			(* Case 51 -  Attesa completamento del comando MOVETOPOS o del raggiungimento quota di Pre-Movimento se abilitata la funzione *)
			51: 
				IF (TipoDiDeposito = DEPOSITO_FALDA_SU_CATASTA AND Programma_Z[55].Stato = INTERROTTO) OR 
				(TipoDiDeposito = DEPOSITO_FALDA_SU_PIAZZOLA AND  Programma_Z[57].Stato = INTERROTTO) THEN
					Ciclo^.Passo := 20;	//NON DOVREBBE ACCADERE									
				ELSE
					IF (TipoDiDeposito = DEPOSITO_FALDA_SU_CATASTA AND Programma_Z[55].Stato = TERMINATO) OR
					(TipoDiDeposito = DEPOSITO_FALDA_SU_PIAZZOLA AND  Programma_Z[57].Stato = TERMINATO)(*OR
						(ModuleAX_Z^.Ax^.Status.ActPosition >= TFProgramma_Ciclo_Falda.Quota_Deposito_Falda_SuPiazzola_Z)*) THEN
						Ciclo^.Passo := 110;
						STEPDone := TRUE;
					END_IF	
				END_IF
				
			(* Case 52 -  Attesa completamento del comando MOVETOPOS o del raggiungimento quota di Pre-Movimento se abilitata la funzione *)
			52: 
				IF Programma_Z[55].Stato = INTERROTTO OR Programma_Z[55].Stato = NON_ESEGUITO OR 
				(TipoDiDeposito = DEPOSITO_FALDA_SU_CATASTA AND Programma_X[52].Stato = INTERROTTO) THEN
					Ciclo^.Passo := 20;	//NON DOVREBBE ACCADERE									
				ELSE
					IF Programma_Z[55].Stato = TERMINATO OR
						(ModuleAX_Z^.Ax^.Status.ActPosition <= Programma^.Quota_StartLenta_Deposito_Falda_SuCatastaPallet_Z + 10) AND Programma_Z[56].Stato = IN_ESECUZIONE THEN
						Ciclo^.Passo := 100;
						STEPDone := TRUE;
					END_IF	
				END_IF	
				
			(* Case 100 - PROGRAMMA[56] ASSE Z -> TRASLAZIONE IN LENTA A QUOTA DI DEPOSITO FALDA SU CATASTA VUOTI  *)
			100:
				IF Programma_Z[55].Stato = INTERROTTO OR
				(TipoDiDeposito = DEPOSITO_FALDA_SU_CATASTA AND  Programma_X[52].Stato = INTERROTTO ) OR
				(TipoDiDeposito = DEPOSITO_FALDA_SU_PIAZZOLA AND (Programma_X[53].Stato = INTERROTTO OR Programma_Z[57].Stato = INTERROTTO)) THEN
					Ciclo^.Passo := 20; //NON DOVREBBE ACCADERE										
				ELSE
					IF StepInto THEN
						Programma_Z[56].Stato := DA_ESEGUIRE;
						Programma_Z[56].InterpolaAsse := NO_INTERPOLAZIONE_ASSE;//FALSE;//NO_INTERPOLAZIONE_ASSE
						ProgrammaToModule_Z := Programma_Z[56];
						Ciclo^.Passo := 101;
						STEPDone := FALSE;
					END_IF
				END_IF
			(* Case 81 -  Attesa completamento del comando MOVETOPOS o del raggiungimento quota di Pre-Movimento se abilitata la funzione *)
			101: 
				IF Programma_Z[56].Stato = INTERROTTO OR 
				(TipoDiDeposito = DEPOSITO_FALDA_SU_CATASTA 	AND NOT Programma_X[52].Stato = TERMINATO) OR
				(TipoDiDeposito = DEPOSITO_FALDA_SU_CATASTA 	AND NOT Programma_Y[52].Stato = TERMINATO) THEN
					Ciclo^.Passo := 20; //NON DOVREBBE ACCADERE										
				ELSE
					IF Programma_Z[56].Stato = TERMINATO THEN
						Ciclo^.Passo := 110;
						STEPDone := TRUE;
					END_IF	
				END_IF
				
			(* Case 110 - UNLOAD MODULO ASPIRAZIONE  *)
			110:
				IF StepInto THEN
					TFParametersArrayClear(ADR(ParametersArray));
					TFCommandSend(CmdUNLOAD,ParametersArray,ModulePinza^.Cmd);
					Ciclo^.Passo := 111;
					STEPDone := FALSE;
				END_IF

			(* Case 71 -  Attesa completamento del comando UNLOAD MODULO ASPIRAZIONE *)
			111: 
				IF TFStateCodeGet(ModulePinza^.State) = StateERROR THEN
					Ciclo^.Passo := 20;
				ELSIF NOT TFStateCodeGet(ModulePinza^.State) = StateUNLOAD_RUN  THEN
					Ciclo^.Passo := 110;										
				ELSE
					IF TFStateCodeGet(ModulePinza^.State) = StateUNLOAD_END THEN
						Ciclo^.Passo := 1000;
						STEPDone := TRUE;
					END_IF	
				END_IF

			(* Case 1000 *)
			1000:
				Ciclo^.Stato := TERMINATO;
				Ciclo^.Passo := 1000;
				
			(* Case 9999 - Ciclo NON annullato o NON terminato*)
			9999:
				Ciclo^.Stato := INTERROTTO;
				Ciclo^.Passo := 9999;
	ELSE						
		;
			
	END_CASE;
ELSE								//Se il ciclo deve essere interrotto, setto il suo nuovo stato
	Ciclo^.Stato := INTERROTTO;
END_IF

END_FUNCTION_BLOCK

// ---- POUs/TFCicliDiLavoro/Lastre/Cicli di Prelievo Lastre/TFCiclo_Prelievo_Lastra.TcPOU
FUNCTION_BLOCK TFCiclo_Prelievo_Lastra
VAR_INPUT
	Ciclo 		: POINTER TO Stato_Ciclo_Lavoro;
	Programma : POINTER TO TFProgramma_Ciclo_Lastra;
	Modules : POINTER TO TFPalletizerModules;
	StartInterpolazioneAssi : POINTER TO BOOL;
	QuotaPassModePuntoIntermedio : ARRAY [1..3] OF REAL;
	AbilitazioneGlobalePassMode	: BOOL;
	InterrompiCiclo : BOOL;
	Abilita_Ciclo_Step : BOOL;
	Command_Step : BOOL;
	AbilitazioneAnticipoDinamicoMovimenti : BOOL;
	PrelievoPezzoOrizzontale : BOOL;//indica che il prelievo del pezzo è orizzontale, sono su pallet o cassa
	NumeroTentativiPresa : UINT := 2;//Numero dei tentativi da effettuare prima di eliminare l'elemento
	InWaitPosition : BOOL; //Macchina in posizione di riposo
	AbilitaLettoreBC : BOOL;//Abilita la lettura del lettore BC
	AbilitaValidazioneLettoreBC : BOOL; //Abilita la validazione del codice letto/non letto dal BC
	Mission : POINTER TO TFMachinePalletizer_Mission;
	//Quota_Rotazione_StartTasteggio_Lastra 		: LREAL;
END_VAR
VAR_OUTPUT
	STEPDone	: BOOL;
	SupportoVuoto : BOOL;
	Errore : UINT;
	BarcodeLetto	: STRING;//Valore del Barcode letto 

END_VAR
VAR
	StepInto : BOOL;
	NumeroTentativiPresaAttuali : UINT;
	TimerAttesaCadutaLastra : REAL;
	i: UINT;
	RichiestaEspulsionePerPolistirolo: BOOL;
	PipickOld : UINT;
	PinzaVerticale	: BOOL;//Indica che la pinza è inclinata e NON in piano, rispetto l'asse J
	AttivazioneVuotoDistanza : BOOL;
	ReqStartAspirazione : BOOL;

	PinzaInPresa : BOOL;
	TimerPartenzaOk : Tc2_Standard.TON;
	QuotaJPerAsseInPiano : LREAL;
	TimerAttesaFiltroFtc : Tc2_Standard.TON;
	PosicionJSalida: LREAL;

	
	PruLineaContactos: BOOL;
END_VAR

//Decido qualce ciclo eseguire
IF Mission^.JPick >= 87 AND Mission^.JPick <= 93 THEN//Se il deposito è a 90 gradi... quindi in orizzontale
	Orizzontale();
ELSE//Se ho deposito in verticale...
	Verticale();
END_IF

ACTION Orizzontale:

TFTimerCall(ADR(TimerAttesaCadutaLastra),TimeBase);
(* Set della variabile che mi permette di fare lo STEP nel ciclo *)
StepInto := (Abilita_Ciclo_Step AND Command_Step) OR NOT Abilita_Ciclo_Step;

(* Reset Anticipo Dinamico se non ho l'abilitazione *)
IF NOT AbilitazioneAnticipoDinamicoMovimenti  OR NOT HMI_DisabilitaAnticipiGLOBALE THEN
	QuotaAnticipoDinamicaX_Raggiunta := FALSE;
	QuotaAnticipoDinamicaY_Raggiunta := FALSE;
	QuotaAnticipoDinamicaZ_Raggiunta := FALSE;
END_IF
PinzaVerticale := Modules^.AX_J.Ax^.Status.ActPosition > 95 OR Modules^.AX_J.Ax^.Status.ActPosition < 85;

PinzaInPresa   := Modules^.Pinza.StatoPinza.ElementoPrelevato OR  
					Modules^.Pinza.StatoPinza.LatoDxPiastrellaInPresa OR
					Modules^.Pinza.StatoPinza.LatoSxPiastrellaInPresa;

IF NOT InterrompiCiclo THEN
	IF Ciclo^.Stato = TERMINATO OR Ciclo^.Stato = ANNULLATO THEN
		Ciclo^.Passo 	:= 0;
		Errore 			:= 0;
	ELSIF Ciclo^.Stato = INTERROTTO THEN
		Ciclo^.Passo 	:= 999;
	ELSE
		Errore := 0;
		Ciclo^.Stato := IN_ESECUZIONE;
	END_IF

	CASE Ciclo^.Passo OF
			(* Case 0 *)
			0:  Ciclo^.Stato 	:= IN_ESECUZIONE;
				Ciclo^.Passo 	:= 10;
				STEPDone 		:= FALSE;
				
			(* Case 10 - Spengo aspirazione *)
			10:	IF Modules^.Pinza.CmdNext.Code = '' AND NOT PinzaInPresa THEN
					TFParametersArrayClear(ADR(ParametersArray));
					TFCommandSend(CmdUNLOAD,ParametersArray,Modules^.Pinza.Cmd);
					Modules^.Pinza.IN.RichiestaRicalibrazioneOvemEsterna := FALSE; //Ricalibrazione automatica OVEM
					Ciclo^.Passo := 20;
				ELSIF PinzaInPresa THEN
					Errore := ErrPRESENZA_MATERIALE_SUPINZA_CICLO_PRELPACCO;
				END_IF

			(* Case 11 - Attesa Aspirazione spenta *)
			11:
				IF TFStateCodeGet(Modules^.Pinza.State) = StateUNLOAD_END THEN
					Ciclo^.Passo := 20;
				END_IF
						
			(* Case 20 - PROGRAMMA[106] ASSE Z -> TRASLAZIONE A QUOTA DI FUORI INGOMBRO *)	
			20:	
				IF StepInto THEN
					IF PinzaVerticale AND NOT AsseXInFinestraDiPrelievo THEN
						Programma_Z[Z_PosFuoriIngombroVuotoLastra].Stato 			:= DA_ESEGUIRE;
						Programma_Z[Z_PosFuoriIngombroVuotoLastra].InterpolaAsse 	:= INTERPOLAZIONE_ASSE;
						ProgrammaToModule_Z 										:= Programma_Z[Z_PosFuoriIngombroVuotoLastra];
						IF Temp_Bool[30] THEN
							Programma_Y[Y_PosFuoriIngombroVuotoLastra].Stato 			:= DA_ESEGUIRE;
							//Programma_Y[Y_PosFuoriIngombroVuotoLastra].InterpolaAsse 	:= INTERPOLAZIONE_ASSE;
							Programma_Y[Y_PosFuoriIngombroVuotoLastra].InterpolaAsse 	:= NO_INTERPOLAZIONE_ASSE;
							ProgrammaToModule_Y 										:= Programma_Y[Y_PosFuoriIngombroVuotoLastra];
						END_IF

						Programma_J[J_PosFuoriIngombro].Stato 			:= DA_ESEGUIRE;
						Programma_J[J_PosFuoriIngombro].InterpolaAsse 	:= INTERPOLAZIONE_ASSE;
						ProgrammaToModule_J 							:= Programma_J[J_PosFuoriIngombro];

						StartInterpolazioneAssi^ 	:= TRUE; //Abilito l'interpolazione degli assi
					ELSE
						Programma_Z[Z_PosFuoriIngombroVuotoLastra].Stato 			:= DA_ESEGUIRE;
						Programma_Z[Z_PosFuoriIngombroVuotoLastra].InterpolaAsse 	:= NO_INTERPOLAZIONE_ASSE;
						ProgrammaToModule_Z 										:= Programma_Z[Z_PosFuoriIngombroVuotoLastra];
					END_IF
					Ciclo^.Passo := 21;
					STEPDone := FALSE;
				END_IF
				
			(* Case 21 - Attesa completamento del comando MOVETOPOS o del raggiungimento quota di Pre-Movimento se abilitata la funzione*)
			21: 
				IF (Programma_Z[Z_PosFuoriIngombroVuotoLastra].Stato = TERMINATO OR
					Asse_Z_InFinestraDiPassMode OR 
					QuotaAnticipoDinamicaZ_Raggiunta)  AND 
					((PinzaVerticale AND NOT AsseXInFinestraDiPrelievo AND
					//(Programma_Y[Y_PosFuoriIngombroVuotoLastra].Stato = TERMINATO OR 
					(Programma_Y[Y_PosFuoriIngombroCaricoLastra].Stato = TERMINATO OR 
					Asse_Y_InFinestraDiPassMode) AND 
					(Programma_J[J_PosFuoriIngombro].Stato = TERMINATO OR 
					Asse_J_InFinestraDiPassMode)) OR NOT PinzaVerticale OR AsseXInFinestraDiPrelievo) THEN
						
						Ciclo^.Passo := 24;
						STEPDone := TRUE;
				ELSIF Programma_Z[Z_PosFuoriIngombroVuotoLastra].Stato = INTERROTTO THEN
					Ciclo^.Passo := 21;										
				END_IF
					
			(* Case 24 - Vado a quota di fuori ingombro y e j  *)
			24:
				IF Programma_Z[Z_PosFuoriIngombroVuotoLastra].Stato = INTERROTTO OR 
					//((PinzaVerticale AND NOT AsseXInFinestraDiPrelievo)AND(Programma_Y[Y_PosFuoriIngombroVuotoLastra].Stato = INTERROTTO OR
					((PinzaVerticale AND NOT AsseXInFinestraDiPrelievo)AND(Programma_Y[Y_PosFuoriIngombroCaricoLastra].Stato = INTERROTTO OR
					Programma_J[J_PosFuoriIngombro].Stato = INTERROTTO)) THEN
						Ciclo^.Passo := 24;										
				ELSE
					IF StepInto THEN
						IF (NOT PinzaVerticale AND NOT AsseXInFinestraDiPrelievo) OR FuoriIngombroYNecessario THEN
							Programma_Y[Y_PosFuoriIngombroVuotoLastra].Stato 			:= DA_ESEGUIRE;
							Programma_Y[Y_PosFuoriIngombroVuotoLastra].InterpolaAsse 	:= INTERPOLAZIONE_ASSE;
							ProgrammaToModule_Y 										:= Programma_Y[Y_PosFuoriIngombroVuotoLastra];
	
							Programma_J[J_PosFuoriIngombro].Stato 			:= DA_ESEGUIRE;
							Programma_J[J_PosFuoriIngombro].InterpolaAsse 	:= INTERPOLAZIONE_ASSE;
							ProgrammaToModule_J 							:= Programma_J[J_PosFuoriIngombro];
							StartInterpolazioneAssi^ 	:= TRUE; //Abilito l'interpolazione degli assi
						END_IF
						IF NOT FuoriIngombroYNecessario THEN
							Programma_X[X_PosStartLentaPrelievoLastra].Stato 			:= DA_ESEGUIRE;
							Programma_X[X_PosStartLentaPrelievoLastra].InterpolaAsse 	:= INTERPOLAZIONE_ASSE;
							ProgrammaToModule_X 										:= Programma_X[X_PosStartLentaPrelievoLastra];
							StartInterpolazioneAssi^ 	:= TRUE; //Abilito l'interpolazione degli assi
							Ciclo^.Passo := 41;
						ELSE
							Ciclo^.Passo := 25;
						END_IF
						STEPDone 					:= FALSE;
					END_IF
				END_IF
				
			(* Case 25 - *)
			25: IF Programma_Z[Z_PosFuoriIngombroVuotoLastra].Stato = INTERROTTO OR  
					(Programma_X[X_PosStartLentaPrelievoLastra].Stato = INTERROTTO AND NOT FuoriIngombroYNecessario) OR
					Programma_Y[Y_PosFuoriIngombroVuotoLastra].Stato = INTERROTTO OR
					Programma_J[J_PosFuoriIngombro].Stato = INTERROTTO THEN
						Ciclo^.Passo := 25;
				ELSIF (Programma_Y[Y_PosFuoriIngombroVuotoLastra].Stato = TERMINATO OR 
					Asse_Y_InFinestraDiPassMode) AND 
					(Programma_J[J_PosFuoriIngombro].Stato = TERMINATO OR 
					Asse_J_InFinestraDiPassMode) THEN	
						Ciclo^.Passo := 40;
						STEPDone := TRUE;	
				END_IF
				
				
			(* Case 40 - PROGRAMMA[] ASSE  -> X TRASLAZIONE A QUOTA DI START LENTA PRELIEVO LASTRA *)	
			40:	
				IF Programma_Z[Z_PosFuoriIngombroVuotoLastra].Stato = INTERROTTO OR
					Programma_Y[Y_PosFuoriIngombroVuotoLastra].Stato = INTERROTTO OR
					Programma_J[J_PosFuoriIngombro].Stato = INTERROTTO THEN
						Ciclo^.Passo := 40;										
				ELSE
					IF StepInto THEN
						Programma_X[X_PosStartLentaPrelievoLastra].Stato 			:= DA_ESEGUIRE;
						Programma_X[X_PosStartLentaPrelievoLastra].InterpolaAsse 	:= NO_INTERPOLAZIONE_ASSE;
						ProgrammaToModule_X 										:= Programma_X[X_PosStartLentaPrelievoLastra];
												
						StartInterpolazioneAssi^ := FALSE; //Abilito l'interpolazione degli assi
						Ciclo^.Passo := 41;
						STEPDone := FALSE;
					END_IF
				END_IF
			
			(* Case 41 -   *)	
			41:	
				IF Programma_Z[Z_PosFuoriIngombroVuotoLastra].Stato = INTERROTTO OR
					(Programma_Y[Y_PosFuoriIngombroVuotoLastra].Stato = INTERROTTO AND FuoriIngombroYNecessario)OR
					(Programma_J[J_PosFuoriIngombro].Stato = INTERROTTO AND FuoriIngombroJNecessario) OR
					Programma_X[X_PosStartLentaPrelievoLastra].Stato = INTERROTTO THEN
						Ciclo^.Passo := 41;										
				ELSE
					STEPDone := TRUE;
					IF StepInto THEN
						Ciclo^.Passo := 42;
						STEPDone := FALSE;
					END_IF
				END_IF
				
			(* Case 42 -  Attesa completamento del comando MOVETOPOS o del raggiungimento quota di Pre-Movimento se abilitata la funzione Y E J IN POS PRELIEVO *)
			42: 
				IF Programma_Z[Z_PosFuoriIngombroVuotoLastra].Stato = INTERROTTO OR
					(Programma_Y[Y_PosFuoriIngombroVuotoLastra].Stato = INTERROTTO AND FuoriIngombroYNecessario)OR
					(Programma_J[J_PosFuoriIngombro].Stato = INTERROTTO AND FuoriIngombroJNecessario) OR
					Programma_X[X_PosStartLentaPrelievoLastra].Stato = INTERROTTO THEN
						Ciclo^.Passo := 42;	
				ELSIF (Programma_X[X_PosStartLentaPrelievoLastra].Stato 	= TERMINATO OR Asse_X_InFinestraDiPassMode) AND
					(Programma_Y[Y_PosFuoriIngombroVuotoLastra].Stato		= TERMINATO OR Asse_Y_InFinestraDiPassMode OR NOT FuoriIngombroYNecessario) AND
					Programma_Z[Z_PosFuoriIngombroVuotoLastra].Stato 		= TERMINATO AND// OR Asse_Z_InFinestraDiPassMode AND
					(Programma_J[J_PosFuoriIngombro].Stato 					= TERMINATO OR Asse_J_InFinestraDiPassMode or not FuoriIngombroJNecessario) THEN
						//Y IN PRELIEVO
						Programma_Y[Y_PosStartLentaPrelievoLastra].Stato 			:= DA_ESEGUIRE;
						Programma_Y[Y_PosStartLentaPrelievoLastra].InterpolaAsse 	:= INTERPOLAZIONE_ASSE;
						ProgrammaToModule_Y 										:= Programma_Y[Y_PosStartLentaPrelievoLastra];
						//J IN PRELIEVO
						Programma_J[J_PosPrelievoLastra].Stato 			:= DA_ESEGUIRE;
						Programma_J[J_PosPrelievoLastra].InterpolaAsse 	:= INTERPOLAZIONE_ASSE;
						ProgrammaToModule_J 							:= Programma_J[J_PosPrelievoLastra];
						StartInterpolazioneAssi^ 						:= TRUE;
						Ciclo^.Passo := 45;
						STEPDone := TRUE;							
				END_IF
				
			(* Case 45 -  *)
			45:
				IF Programma_Z[Z_PosFuoriIngombroVuotoLastra].Stato = INTERROTTO OR
					Programma_Y[Y_PosStartLentaPrelievoLastra].Stato = INTERROTTO OR
					Programma_J[J_PosPrelievoLastra].Stato = INTERROTTO OR
					Programma_X[X_PosStartLentaPrelievoLastra].Stato = INTERROTTO THEN
						Ciclo^.Passo := 45;	
				ELSIF (Programma_X[X_PosStartLentaPrelievoLastra].Stato 	= TERMINATO OR Asse_X_InFinestraDiPassMode) AND
					(Programma_Y[Y_PosStartLentaPrelievoLastra].Stato		= TERMINATO OR Asse_Y_InFinestraDiPassMode) AND
					Programma_Z[Z_PosFuoriIngombroVuotoLastra].Stato 		= TERMINATO AND// OR Asse_Z_InFinestraDiPassMode AND
					(Programma_J[J_PosPrelievoLastra].Stato 				= TERMINATO OR Asse_J_InFinestraDiPassMode) THEN
						Ciclo^.Passo := 50;
				END_IF
							
			(* Case 50 - PROGRAMMA[101] ASSE Z -> TRASLAZIONE A QUOTA AMMESSA IN VELOCE DI PRELIEVO PACCO  *)
			50:	
				///IF Programma_Z[Z_PosFuoriIngombroVuotoLastra].Stato = INTERROTTO OR
				///	Programma_Y[Y_PosStartLentaPrelievoLastra].Stato = INTERROTTO OR
				///	Programma_J[J_PosPrelievoLastra].Stato = INTERROTTO OR
				///	Programma_X[X_PosStartLentaPrelievoLastra].Stato = INTERROTTO THEN
				///		Ciclo^.Passo := 50;	
				///ELSIF (Programma_X[X_PosStartLentaPrelievoLastra].Stato 	= TERMINATO OR Asse_X_InFinestraDiPassMode) AND
				///	(Programma_Y[Y_PosStartLentaPrelievoLastra].Stato		= TERMINATO OR Asse_Y_InFinestraDiPassMode) AND
				///	Programma_Z[Z_PosFuoriIngombroVuotoLastra].Stato 		= TERMINATO AND// OR Asse_Z_InFinestraDiPassMode AND
				///	(Programma_J[J_PosPrelievoLastra].Stato 				= TERMINATO OR Asse_J_InFinestraDiPassMode) AND
				IF StepInto THEN
					Programma_Z[Z_PosStartLentaPrelievoLastra].Stato 			:= DA_ESEGUIRE;
					Programma_Z[Z_PosStartLentaPrelievoLastra].InterpolaAsse 	:= NO_INTERPOLAZIONE_ASSE;
					ProgrammaToModule_Z 										:= Programma_Z[Z_PosStartLentaPrelievoLastra];
					Ciclo^.Passo := 51;
					STEPDone := FALSE;
				END_IF
				

			(* Case 51 -  Attesa completamento del comando MOVETOPOS o del raggiungimento quota di Pre-Movimento se abilitata la funzione *)
			51: 
				IF Programma_Z[Z_PosStartLentaPrelievoLastra].Stato = INTERROTTO OR
					Programma_Y[Y_PosStartLentaPrelievoLastra].Stato = INTERROTTO OR
					Programma_J[J_PosFuoriIngombro].Stato = INTERROTTO OR
					Programma_X[X_PosStartLentaPrelievoLastra].Stato = INTERROTTO THEN
						Ciclo^.Passo := 51;									
				ELSE
					IF Programma_X[X_PosStartLentaPrelievoLastra].Stato 	= TERMINATO AND
						Programma_Y[Y_PosStartLentaPrelievoLastra].Stato	= TERMINATO AND
						Programma_J[J_PosPrelievoLastra].Stato 				= TERMINATO AND
						(Programma_Z[Z_PosStartLentaPrelievoLastra].Stato = TERMINATO OR 
						(Modules^.AX_Z.Ax^.Status.ActPosition <= Programma_Z[Z_PosStartLentaPrelievoLastra].Quota_Destinazione + 10)) THEN
							Ciclo^.Passo := 90;
							STEPDone := TRUE;
					END_IF	
				END_IF

			(* Case 90 - ATTIVAZIONE ASPIRAZIONE *)
			90:
				IF Programma_Z[Z_PosStartLentaPrelievoLastra].Stato = INTERROTTO THEN
					Ciclo^.Passo := 90; 									
				ELSE
					IF StepInto THEN
						TFParametersArrayClear(ADR(ParametersArray));
						ParametersArray.Parameters[0] := BOOL_TO_STRING(NOT PrelievoPezzoOrizzontale);//SE TRUE: pezzo prelevato da cavallina, altrimenti prelievo orizzontale
						ParametersArray.Parameters[1] := BOOL_TO_STRING(FALSE);//SE TRUE: ATTIVO SOLO VENTOSE CARTONE
						TFCommandSend(CmdPRELOAD,ParametersArray,Modules^.Pinza.Cmd);//LANCIO COMANDO ASPIRAZIONE PINZA
						Ciclo^.Passo := 91;
						STEPDone := FALSE;
					END_IF
				END_IF	
	
			(* Case 91 -  Attesa completamento dei comandi *)
			91: 
				IF TFStateCodeGet(Modules^.Pinza.State) = StateERROR THEN //Modulo pinza in errore
					Ciclo^.Passo := 91; 										
				ELSE
					IF TFStateCodeGet(Modules^.Pinza.State) = StatePRELOAD_END THEN //Aspirazione in corso 
						Ciclo^.Passo := 100;
						STEPDone := FALSE;
					END_IF	
				END_IF
				
			(* Case 100 - FREE *)
			100:
				Ciclo^.Passo := 101;
			(* Case 101 - FREE *)
			101: 
				Ciclo^.Passo := 150;
				
			(* Case 150 - Tasteggio in direzione Z *)
			150: 
				IF Programma_Z[Z_PosStartLentaPrelievoLastra].Stato = INTERROTTO THEN
					Ciclo^.Passo := 150;									
				ELSE
					IF StepInto THEN
						Programma_Z[Z_PosPrelievoInLentaLastra].Stato 			:= DA_ESEGUIRE;
						Programma_Z[Z_PosPrelievoInLentaLastra].InterpolaAsse 	:= NO_INTERPOLAZIONE_ASSE;
						ProgrammaToModule_Z 									:= Programma_Z[Z_PosPrelievoInLentaLastra];
	
						Ciclo^.Passo := 155;
						STEPDone := FALSE;
					END_IF	
				END_IF
		
			(* Case 155 - VADO A ESEGUIRE IL DISTACCO LASTRA *)
			155: 
				IF Programma_Z[Z_PosPrelievoInLentaLastra].Stato = INTERROTTO THEN
						Ciclo^.Passo := 155;																
				ELSE
					IF Programma_Z[Z_PosPrelievoInLentaLastra].Stato = TERMINATO THEN
						Ciclo^.Passo 	:= 156;
						Programma_Z[Z_PosDistaccoLastraInLentaLastra].Quota_Destinazione := Modules^.AX_Z.QuotaAsseLetturaTasteggio + OffsetDistacco.Lastra.Z;
						//	
										
						STEPDone := TRUE;
					END_IF	
				END_IF

			(* Case 156 - Distacco lastra *)
			156: 
				IF StepInto THEN
					Programma_Z[Z_PosDistaccoLastraInLentaLastra].Stato 			:= DA_ESEGUIRE;
					Programma_Z[Z_PosDistaccoLastraInLentaLastra].InterpolaAsse 	:= NO_INTERPOLAZIONE_ASSE;
					ProgrammaToModule_Z 											:= Programma_Z[Z_PosDistaccoLastraInLentaLastra];
								
					Ciclo^.Passo := 157;
					STEPDone := FALSE;
				END_IF	

